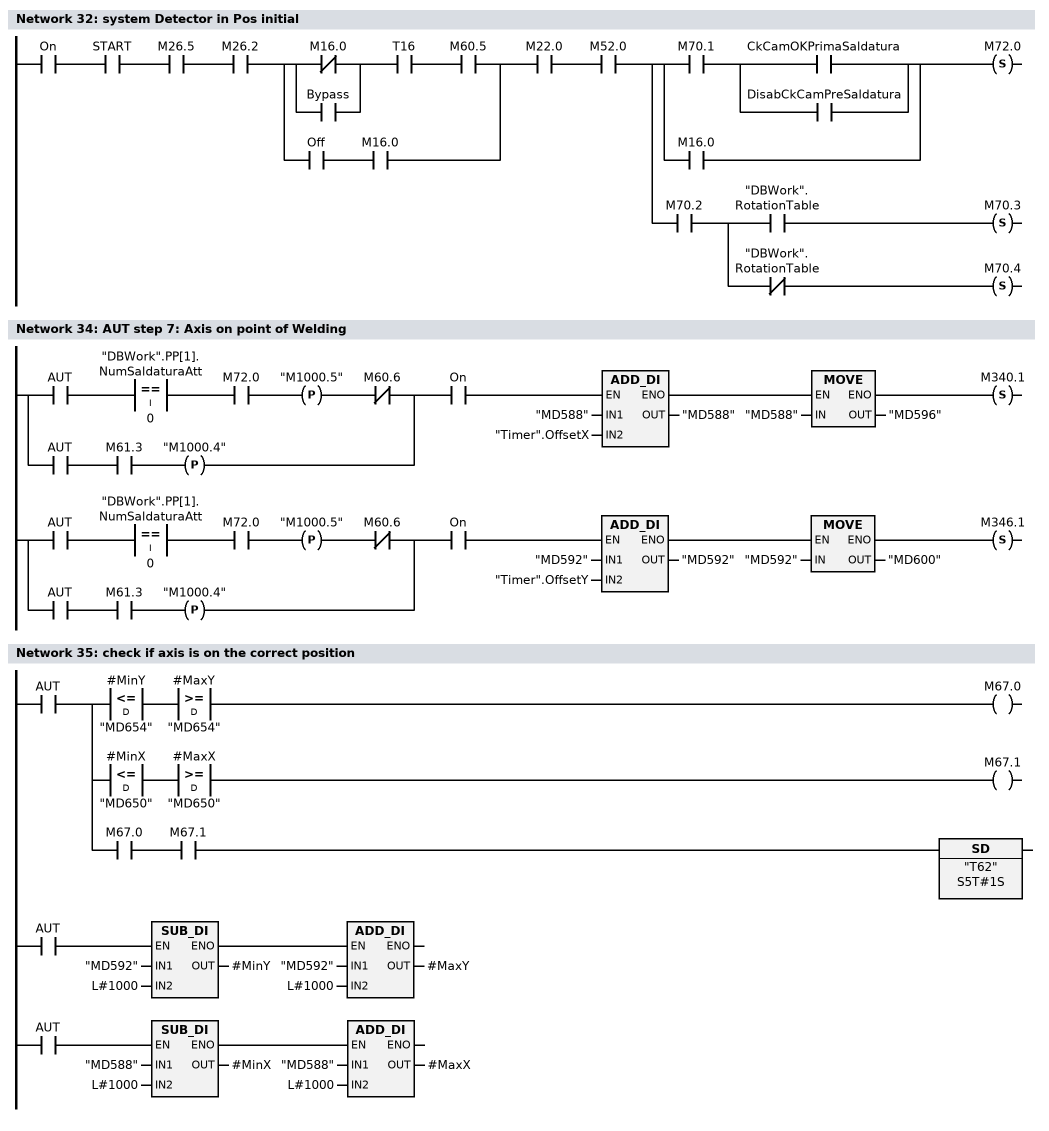
[picture p121: FC14 - AUTOMATIC networks 32-35]
NETWORK
TITLE = system Detector in Pos initial
//System Detector in Pos initial and ready for detect Welding point
      A     "On";
      A     "START";
      A     "M26.5";
      A     "M26.2";
      A(;
      A(;
      ON    "M16.0";
      O     "Bypass";
      );
      A     "T16";
      A     "M60.5";
      O;
      A     "Off";
      A     "M16.0";
      );
      A     "M22.0";
      A     "M52.0";
      =     L 16.0;
      A     L 16.0;
      A(;
      A     "M70.1";
      A(;
      O     "CkCamOKPrimaSaldatura";
      O     "DisabCkCamPreSaldatura";
      );
      O     "M16.0";
      );
      S     "M72.0";
      A     L 16.0;
      A     "M70.2";
      =     L 16.1;
      A     L 16.1;
      A     "DBWork".RotationTable;
      S     "M70.3";
      A     L 16.1;
      AN    "DBWork".RotationTable;
      S     "M70.4";
NETWORK
TITLE = ------------START WITH WELDING
NETWORK
TITLE = AUT step 7: Axis on point of Welding
//AXIS X 
//AXIS Y 
//
//MD588 = SUPPORT FOR POINT X
//MD592 = SUPPORT FOR POINT Y
      A(;
      A     "AUT";
      A(;
      L     "DBWork".PP[1].NumSaldaturaAtt;
      L     0;
      ==I;
      );
      A     "M72.0";
      FP    "M1000.5";
      AN    "M60.6";
      O(;
      A     "AUT";
      A     "M61.3";
      FP    "M1000.4";
      );
      );
      A     "On";
      =     L 16.0;
      A(;
      A     L 16.0;
      JNB   _018;
      L     "MD588";
      L     "Timer".OffsetX;
      +D;
      T     "MD588";
      AN    OV;
      SAVE;
      CLR;
_018: A     BR;
      );
      JNB   _019;
      L     "MD588";
      T     "MD596";
      SET;
      SAVE;
      CLR;
_019: A     BR;
      S     "M340.1";
      A(;
      A     L 16.0;
      JNB   _01a;
      L     "MD592";
      L     "Timer".OffsetY;
      +D;
      T     "MD592";
      AN    OV;
      SAVE;
      CLR;
_01a: A     BR;
      );
      JNB   _01b;
      L     "MD592";
      T     "MD600";
      SET;
      SAVE;
      CLR;
_01b: A     BR;
      S     "M346.1";
NETWORK
TITLE = check if axis is on the correct position
      A     "AUT";
      =     L 16.0;
      A(;
      A     L 16.0;
      JNB   _01c;
      L     "MD592";
      L     L#1000;
      -D;
      T     #MinY;
      AN    OV;
      SAVE;
      CLR;
_01c: A     BR;
      );
      JNB   _01d;
      L     "MD592";
      L     L#1000;
      +D;
      T     #MaxY;
_01d: NOP   0;
      A(;
      A     L 16.0;
      JNB   _01e;
      L     "MD588";
      L     L#1000;
      -D;
      T     #MinX;
      AN    OV;
      SAVE;
      CLR;
_01e: A     BR;
      );
      JNB   _01f;
      L     "MD588";
      L     L#1000;
      +D;
      T     #MaxX;
_01f: NOP   0;
      A     L 16.0;
      A(;
      L     #MinY;
      L     "MD654";
      <=D;
      );
      A(;
      L     #MaxY;
      L     "MD654";
      >=D;
      );
      =     "M67.0";
      A     L 16.0;
      A(;
      L     #MinX;
      L     "MD650";
      <=D;
      );
      A(;
      L     #MaxX;
      L     "MD650";
      >=D;
      );
      =     "M67.1";
      A     L 16.0;
      A     "M67.0";
      A     "M67.1";
      L     S5T#1S;
      SD    "T62";
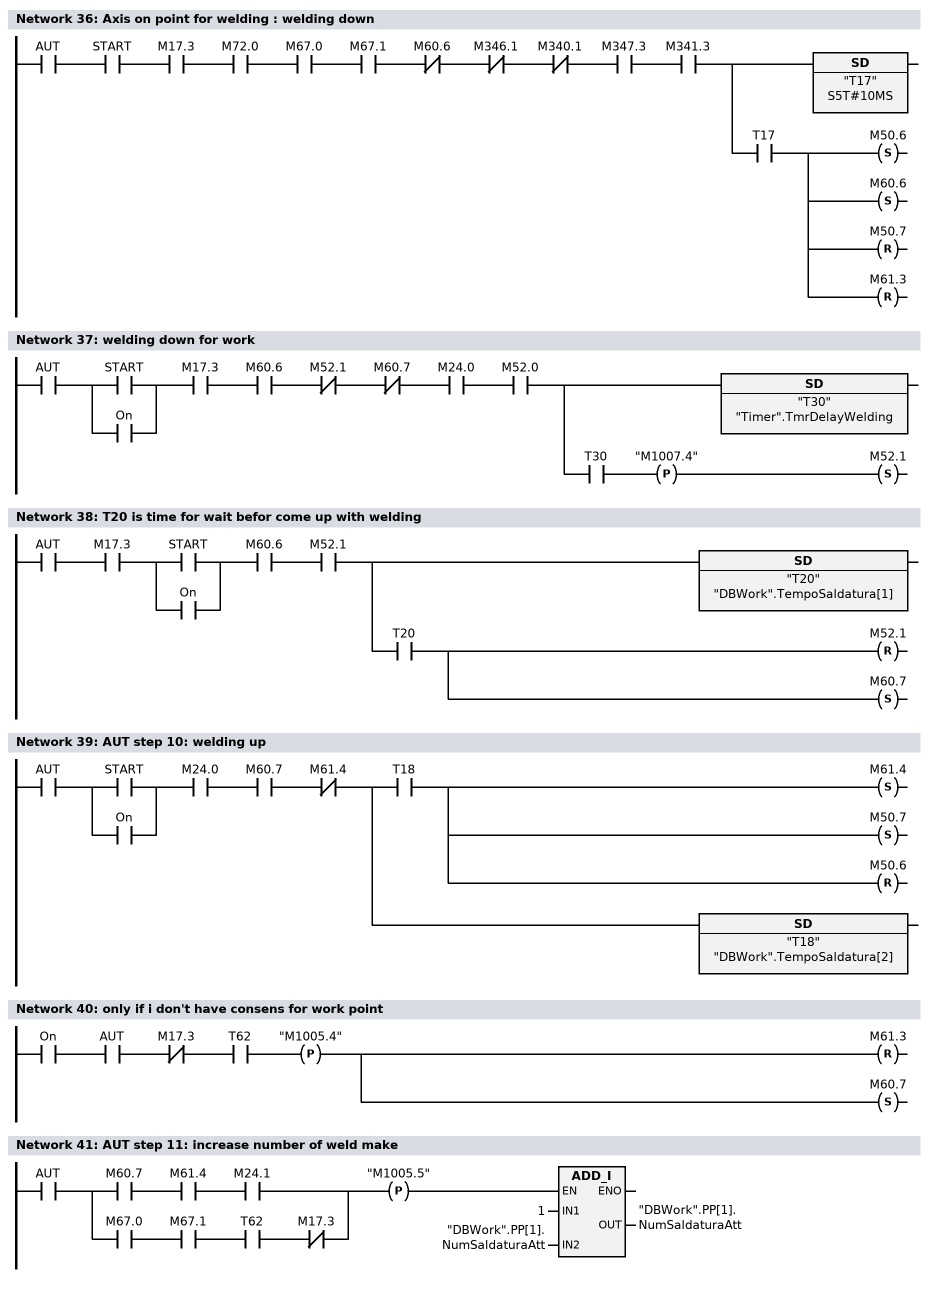
NETWORK
TITLE = Axis on point for welding : welding down
//Saldatore giù
      A     "AUT";
      A     "START";
      A     "M17.3";
      A     "M72.0";
      A     "M67.0";
      A     "M67.1";
      AN    "M60.6";
      AN    "M346.1";
      AN    "M340.1";
      A     "M347.3";
      A     "M341.3";
      =     L 16.0;
      A     L 16.0;
      BLD   102;
      L     S5T#10MS;
      SD    "T17";
      A     L 16.0;
      A     "T17";
      S     "M50.6";
      S     "M60.6";
      R     "M50.7";
      R     "M61.3";
NETWORK
TITLE = welding down for work
//saldatore giu per saldatura
      A     "AUT";
      A(;
      O     "START";
      O     "On";
      );
      A     "M17.3";
      A     "M60.6";
      AN    "M52.1";
      AN    "M60.7";
      A     "M24.0";
      A     "M52.0";
      =     L 16.0;
      A     L 16.0;
      BLD   102;
      L     "Timer".TmrDelayWelding;
      SD    "T30";
      A     L 16.0;
      A     "T30";
      FP    "M1007.4";
      S     "M52.1";
NETWORK
TITLE = T20 is time for wait befor come up with welding
//Resto un tempo T20 sul punto saldato prima di rialzare la torcia
      A     "AUT";
      A     "M17.3";
      A(;
      O     "START";
      O     "On";
      );
      A     "M60.6";
      A     "M52.1";
      =     L 16.0;
      A     L 16.0;
      BLD   102;
      L     "DBWork".TempoSaldatura[1];
      SD    "T20";
      A     L 16.0;
      A     "T20";
      R     "M52.1";
      S     "M60.7";
NETWORK
TITLE = AUT step 10: welding up
      A     "AUT";
      A(;
      O     "START";
      O     "On";
      );
      A     "M24.0";
      A     "M60.7";
      AN    "M61.4";
      =     L 16.0;
      A     L 16.0;
      A     "T18";
      S     "M61.4";
      S     "M50.7";
      R     "M50.6";
      A     L 16.0;
      BLD   102;
      L     "DBWork".TempoSaldatura[2];
      SD    "T18";
NETWORK
TITLE = only if i don't have consens for work point
      A     "On";
      A     "AUT";
      AN    "M17.3";
      A     "T62";
      FP    "M1005.4";
      R     "M61.3";
      S     "M60.7";
NETWORK
TITLE = AUT step 11: increase number of weld make
//incremento il numero di saldature effettuate
      A     "AUT";
      A(;
      A     "M60.7";
      A     "M61.4";
      A     "M24.1";
      O;
      A     "M67.0";
      A     "M67.1";
      A     "T62";
      AN    "M17.3";
      );
      FP    "M1005.5";
      JNB   _020;
      L     1;
      L     "DBWork".PP[1].NumSaldaturaAtt;
      +I;
      T     "DBWork".PP[1].NumSaldaturaAtt;
_020: NOP   0;
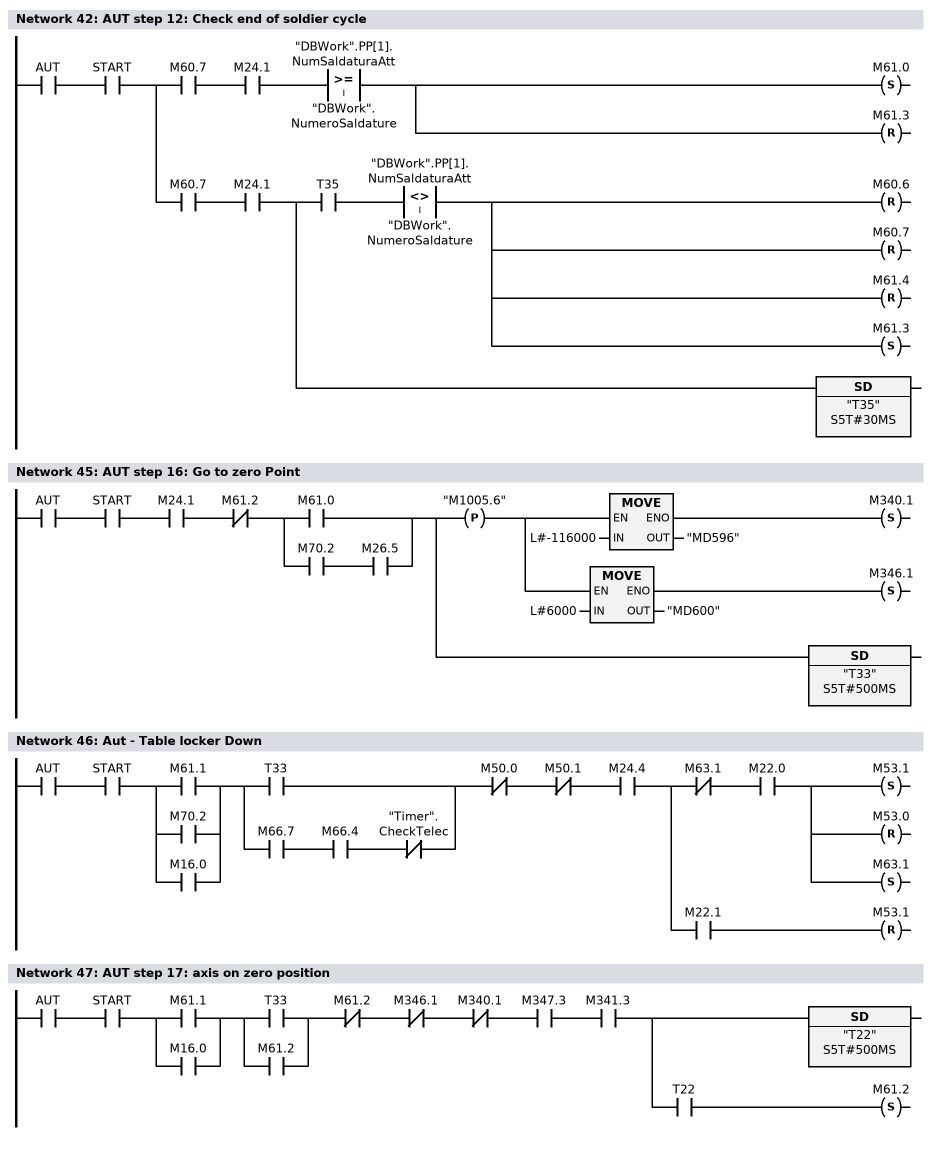
NETWORK
TITLE = AUT step 12: Check end of soldier cycle 
//aspetto per il passaggio delle coorddinate al simodrive
      A     "AUT";
      A     "START";
      =     L 16.0;
      A     L 16.0;
      A     "M60.7";
      A     "M24.1";
      A(;
      L     "DBWork".PP[1].NumSaldaturaAtt;
      L     "DBWork".NumeroSaldature;
      >=I;
      );
      S     "M61.0";
      R     "M61.3";
      A     L 16.0;
      A     "M60.7";
      A     "M24.1";
      =     L 16.1;
      A     L 16.1;
      A     "T35";
      A(;
      L     "DBWork".PP[1].NumSaldaturaAtt;
      L     "DBWork".NumeroSaldature;
      <>I;
      );
      R     "M60.6";
      R     "M60.7";
      R     "M61.4";
      S     "M61.3";
      A     L 16.1;
      BLD   102;
      L     S5T#30MS;
      SD    "T35";
NETWORK
TITLE =
NETWORK
TITLE =
NETWORK
TITLE = AUT step 16: Go to zero Point
      A     "AUT";
      A     "START";
      A     "M24.1";
      AN    "M61.2";
      A(;
      O     "M61.0";
      O;
      A     "M70.2";
      A     "M26.5";
      );
      =     L 16.0;
      A     L 16.0;
      FP    "M1005.6";
      =     L 16.1;
      A     L 16.1;
      JNB   _021;
      L     L#-116000;
      T     "MD596";
      SET;
      SAVE;
      CLR;
_021: A     BR;
      S     "M340.1";
      A     L 16.1;
      JNB   _022;
      L     L#6000;
      T     "MD600";
      SET;
      SAVE;
      CLR;
_022: A     BR;
      S     "M346.1";
      A     L 16.0;
      BLD   102;
      L     S5T#500MS;
      SD    "T33";
NETWORK
TITLE = Aut - Table locker Down
//Table cyclinder Low
      A     "AUT";
      A     "START";
      A(;
      O     "M61.1";
      O     "M70.2";
      O     "M16.0";
      );
      A(;
      O     "T33";
      O;
      A     "M66.7";
      A     "M66.4";
      AN    "Timer".CheckTelec;
      );
      AN    "M50.0";
      AN    "M50.1";
      A     "M24.4";
      =     L 16.0;
      A     L 16.0;
      AN    "M63.1";
      A     "M22.0";
      S     "M53.1";
      R     "M53.0";
      S     "M63.1";
      A     L 16.0;
      A     "M22.1";
      R     "M53.1";
NETWORK
TITLE = AUT step 17: axis on zero position
      A     "AUT";
      A     "START";
      A(;
      O     "M61.1";
      O     "M16.0";
      );
      A(;
      O     "T33";
      O     "M61.2";
      );
      AN    "M61.2";
      AN    "M346.1";
      AN    "M340.1";
      A     "M347.3";
      A     "M341.3";
      =     L 16.0;
      A     L 16.0;
      BLD   102;
      L     S5T#500MS;
      SD    "T22";
      A     L 16.0;
      A     "T22";
      S     "M61.2";
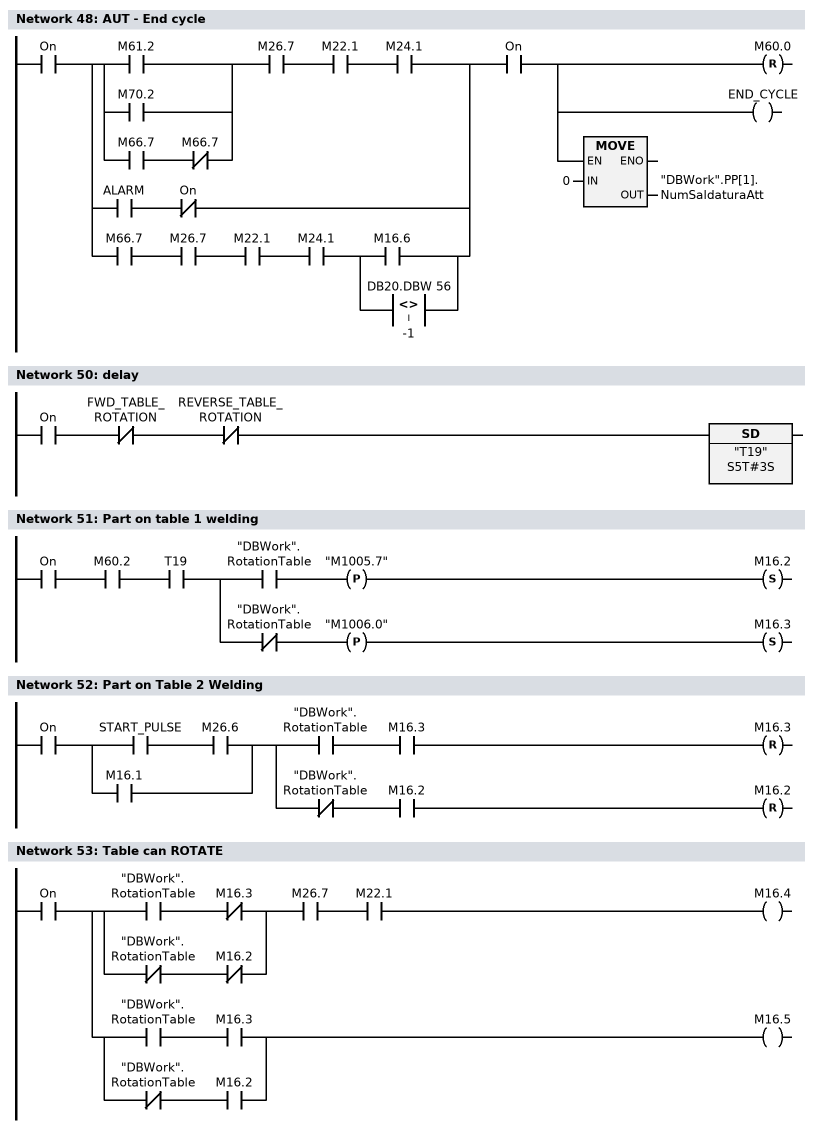
NETWORK
TITLE = AUT - End cycle
      A     "On";
      A(;
      A(;
      O     "M61.2";
      O     "M70.2";
      O;
      A     "M66.7";
      AN    "M66.7";
      );
      A     "M26.7";
      A     "M22.1";
      A     "M24.1";
      O;
      A     "ALARM";
      AN    "On";
      O;
      A     "M66.7";
      A     "M26.7";
      A     "M22.1";
      A     "M24.1";
      A(;
      O     "M16.6";
      O(;
      L     DB20.DBW 56;
      L     -1;
      <>I;
      );
      );
      );
      A     "On";
      =     L 16.0;
      A     L 16.0;
      BLD   102;
      R     "M60.0";
      A     L 16.0;
      BLD   102;
      =     "END_CYCLE";
      A     L 16.0;
      JNB   _023;
      L     0;
      T     "DBWork".PP[1].NumSaldaturaAtt;
_023: NOP   0;
NETWORK
TITLE =
NETWORK
TITLE = delay
      A     "On";
      AN    "FWD_TABLE_ROTATION";
      AN    "REVERSE_TABLE_ROTATION";
      L     S5T#3S;
      SD    "T19";
NETWORK
TITLE = Part on table 1 welding
      A     "On";
      A     "M60.2";
      A     "T19";
      =     L 16.0;
      A     L 16.0;
      A     "DBWork".RotationTable;
      FP    "M1005.7";
      S     "M16.2";
      A     L 16.0;
      AN    "DBWork".RotationTable;
      FP    "M1006.0";
      S     "M16.3";
NETWORK
TITLE = Part on Table 2 Welding
      A     "On";
      A(;
      A     "START_PULSE";
      A     "M26.6";
      O     "M16.1";
      );
      =     L 16.0;
      A     L 16.0;
      A     "DBWork".RotationTable;
      A     "M16.3";
      R     "M16.3";
      A     L 16.0;
      AN    "DBWork".RotationTable;
      A     "M16.2";
      R     "M16.2";
NETWORK
TITLE = Table can ROTATE
      A     "On";
      =     L 16.0;
      A     L 16.0;
      A(;
      A     "DBWork".RotationTable;
      AN    "M16.3";
      O;
      AN    "DBWork".RotationTable;
      AN    "M16.2";
      );
      A     "M26.7";
      A     "M22.1";
      =     "M16.4";
      A     L 16.0;
      A(;
      A     "DBWork".RotationTable;
      A     "M16.3";
      O;
      AN    "DBWork".RotationTable;
      A     "M16.2";
      );
      =     "M16.5";
END_FUNCTION

FUNCTION "FC16 - ALARMS" : VOID	// FC 16
TITLE = Alarms management
VERSION : 0.1
VAR_TEMP
  tempBOOL : BOOL ;
END_VAR
BEGIN
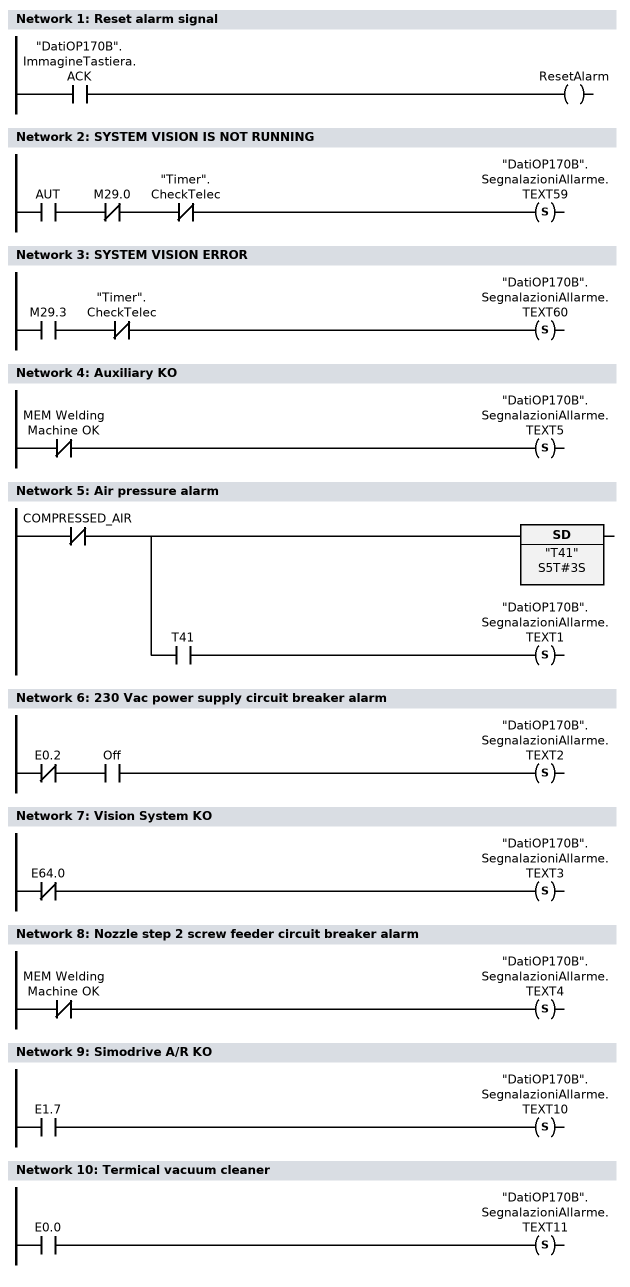
NETWORK
TITLE = Reset alarm signal
      A     "DatiOP170B".ImmagineTastiera.ACK;
      =     "ResetAlarm";
NETWORK
TITLE = SYSTEM VISION IS NOT RUNNING
      A     "AUT";
      AN    "M29.0";
      AN    "Timer".CheckTelec;
      S     "DatiOP170B".SegnalazioniAllarme.TEXT59;
NETWORK
TITLE = SYSTEM VISION ERROR
      A     "M29.3";
      AN    "Timer".CheckTelec;
      S     "DatiOP170B".SegnalazioniAllarme.TEXT60;
NETWORK
TITLE = Auxiliary KO
      AN    "MEM Welding Machine OK";
      S     "DatiOP170B".SegnalazioniAllarme.TEXT5;
NETWORK
TITLE = Air pressure alarm
      AN    "COMPRESSED_AIR";
      =     L 1.0;
      A     L 1.0;
      BLD   102;
      L     S5T#3S;
      SD    "T41";
      A     L 1.0;
      A     "T41";
      S     "DatiOP170B".SegnalazioniAllarme.TEXT1;
NETWORK
TITLE = 230 Vac power supply circuit breaker alarm
      AN    "E0.2";
      A     "Off";
      S     "DatiOP170B".SegnalazioniAllarme.TEXT2;
NETWORK
TITLE = Vision System KO
      AN    "E64.0";
      S     "DatiOP170B".SegnalazioniAllarme.TEXT3;
NETWORK
TITLE = Nozzle step 2 screw feeder circuit breaker alarm
      AN    "MEM Welding Machine OK";
      S     "DatiOP170B".SegnalazioniAllarme.TEXT4;
NETWORK
TITLE = Simodrive A/R KO
      A     "E1.7";
      S     "DatiOP170B".SegnalazioniAllarme.TEXT10;
NETWORK
TITLE = Termical vacuum cleaner
      A     "E0.0";
      S     "DatiOP170B".SegnalazioniAllarme.TEXT11;
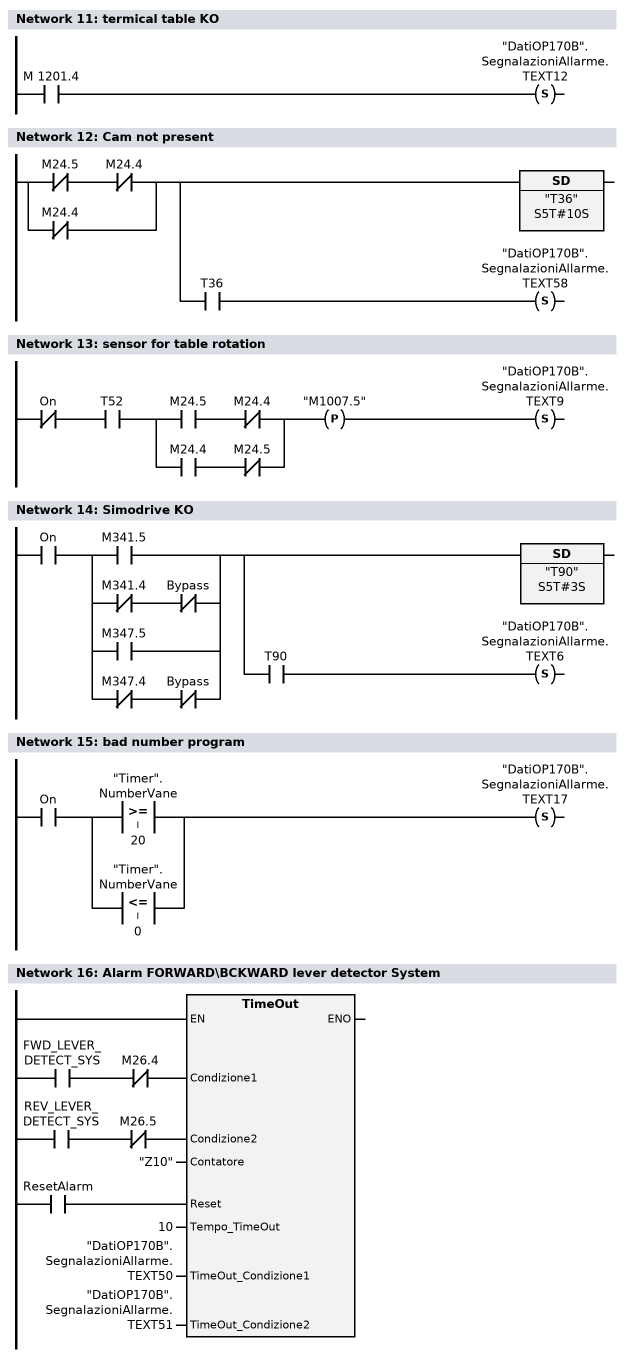
NETWORK
TITLE = termical table KO
      A     M 1201.4;
      S     "DatiOP170B".SegnalazioniAllarme.TEXT12;
NETWORK
TITLE = Cam not present
      AN    "M24.5";
      AN    "M24.4";
      ON    "M24.4";
      =     L 1.0;
      A     L 1.0;
      BLD   102;
      L     S5T#10S;
      SD    "T36";
      A     L 1.0;
      A     "T36";
      S     "DatiOP170B".SegnalazioniAllarme.TEXT58;
NETWORK
TITLE = sensor for table rotation
      AN    "On";
      A     "T52";
      A(;
      A     "M24.5";
      AN    "M24.4";
      O;
      A     "M24.4";
      AN    "M24.5";
      );
      FP    "M1007.5";
      S     "DatiOP170B".SegnalazioniAllarme.TEXT9;
NETWORK
TITLE = Simodrive KO
//press ack button
      A     "On";
      A(;
      O     "M341.5";
      O;
      AN    "M341.4";
      AN    "Bypass";
      O     "M347.5";
      O;
      AN    "M347.4";
      AN    "Bypass";
      );
      =     L 1.0;
      A     L 1.0;
      BLD   102;
      L     S5T#3S;
      SD    "T90";
      A     L 1.0;
      A     "T90";
      S     "DatiOP170B".SegnalazioniAllarme.TEXT6;
NETWORK
TITLE = bad number program
      A     "On";
      A(;
      O(;
      L     "Timer".NumberVane;
      L     20;
      >=I;
      );
      O(;
      L     "Timer".NumberVane;
      L     0;
      <=I;
      );
      );
      S     "DatiOP170B".SegnalazioniAllarme.TEXT17;
NETWORK
TITLE = Alarm FORWARD\BCKWARD lever detector System
      A     "FWD_LEVER_DETECT_SYS";
      AN    "M26.4";
      =     L 1.0;
      BLD   103;
      A     "REV_LEVER_DETECT_SYS";
      AN    "M26.5";
      =     L 1.1;
      BLD   103;
      A     "ResetAlarm";
      =     L 1.2;
      BLD   103;
      CALL  "TimeOut" (
           Condizione1              := L 1.0,
           Condizione2              := L 1.1,
           Contatore                := "Z10",
           Reset                    := L 1.2,
           Tempo_TimeOut            := 10,
           TimeOut_Condizione1      := "DatiOP170B".SegnalazioniAllarme.TEXT50,
           TimeOut_Condizione2      := "DatiOP170B".SegnalazioniAllarme.TEXT51);
      NOP   0;
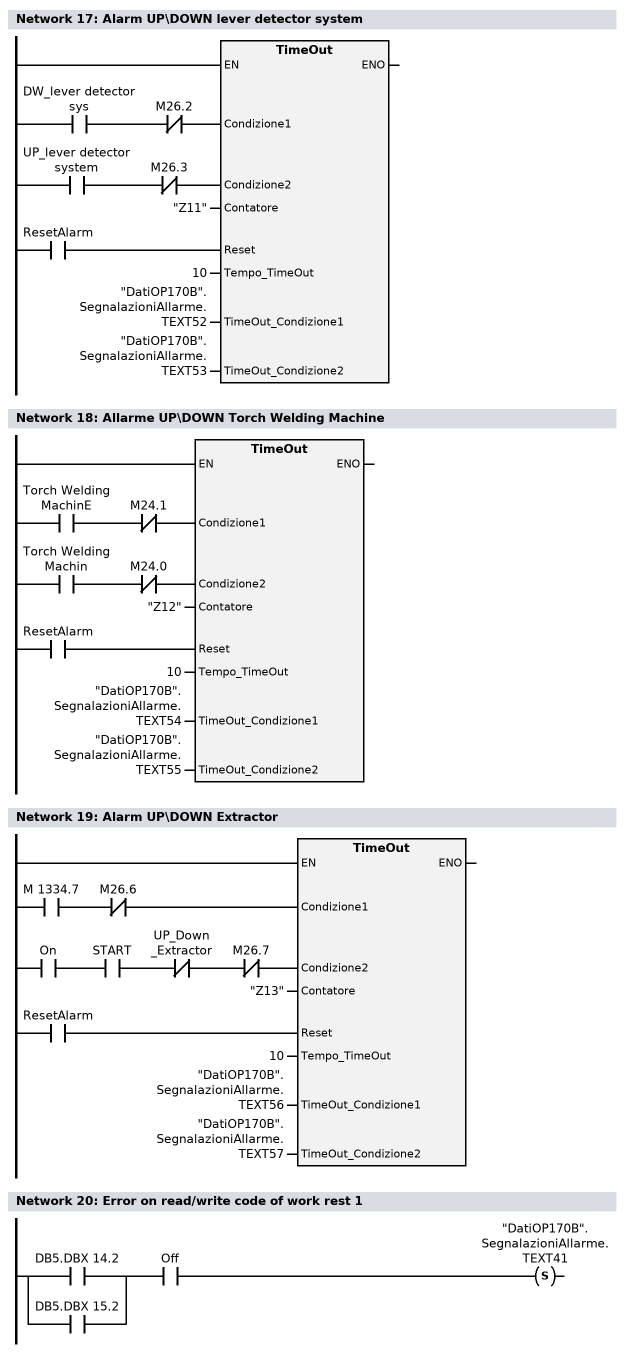
NETWORK
TITLE = Alarm UP\DOWN lever detector system
      A     "DW_lever detector sys";
      AN    "M26.2";
      =     L 1.0;
      BLD   103;
      A     "UP_lever detector system";
      AN    "M26.3";
      =     L 1.1;
      BLD   103;
      A     "ResetAlarm";
      =     L 1.2;
      BLD   103;
      CALL  "TimeOut" (
           Condizione1              := L 1.0,
           Condizione2              := L 1.1,
           Contatore                := "Z11",
           Reset                    := L 1.2,
           Tempo_TimeOut            := 10,
           TimeOut_Condizione1      := "DatiOP170B".SegnalazioniAllarme.TEXT52,
           TimeOut_Condizione2      := "DatiOP170B".SegnalazioniAllarme.TEXT53);
      NOP   0;
NETWORK
TITLE = Allarme UP\DOWN Torch Welding Machine
      A     "Torch Welding MachinE";
      AN    "M24.1";
      =     L 1.0;
      BLD   103;
      A     "Torch Welding Machin";
      AN    "M24.0";
      =     L 1.1;
      BLD   103;
      A     "ResetAlarm";
      =     L 1.2;
      BLD   103;
      CALL  "TimeOut" (
           Condizione1              := L 1.0,
           Condizione2              := L 1.1,
           Contatore                := "Z12",
           Reset                    := L 1.2,
           Tempo_TimeOut            := 10,
           TimeOut_Condizione1      := "DatiOP170B".SegnalazioniAllarme.TEXT54,
           TimeOut_Condizione2      := "DatiOP170B".SegnalazioniAllarme.TEXT55);
      NOP   0;
NETWORK
TITLE = Alarm UP\DOWN Extractor
      A     M 1334.7;
      AN    "M26.6";
      =     L 1.0;
      BLD   103;
      A     "On";
      A     "START";
      AN    "UP_Down _Extractor";
      AN    "M26.7";
      =     L 1.1;
      BLD   103;
      A     "ResetAlarm";
      =     L 1.2;
      BLD   103;
      CALL  "TimeOut" (
           Condizione1              := L 1.0,
           Condizione2              := L 1.1,
           Contatore                := "Z13",
           Reset                    := L 1.2,
           Tempo_TimeOut            := 10,
           TimeOut_Condizione1      := "DatiOP170B".SegnalazioniAllarme.TEXT56,
           TimeOut_Condizione2      := "DatiOP170B".SegnalazioniAllarme.TEXT57);
      NOP   0;
NETWORK
TITLE = Error on read/write code of work rest 1
      A(;
      O     DB5.DBX 14.2;
      O     DB5.DBX 15.2;
      );
      A     "Off";
      S     "DatiOP170B".SegnalazioniAllarme.TEXT41;
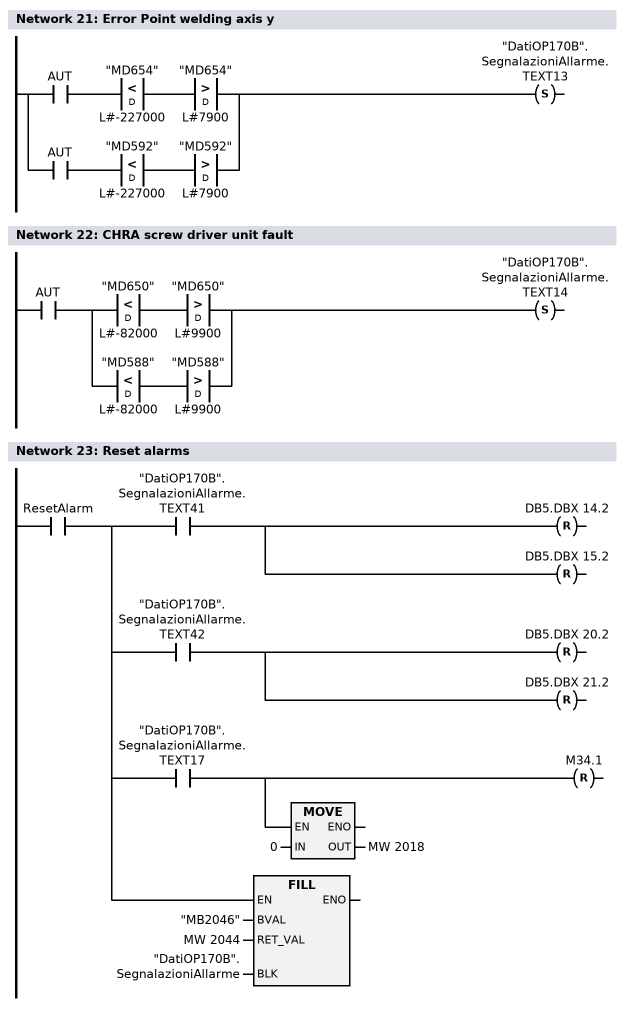
NETWORK
TITLE = Error Point welding axis y
      A     "AUT";
      A(;
      L     "MD654";
      L     L#-227000;
      <D;
      );
      A(;
      L     "MD654";
      L     L#7900;
      >D;
      );
      O;
      A     "AUT";
      A(;
      L     "MD592";
      L     L#-227000;
      <D;
      );
      A(;
      L     "MD592";
      L     L#7900;
      >D;
      );
      S     "DatiOP170B".SegnalazioniAllarme.TEXT13;
NETWORK
TITLE = CHRA screw driver unit fault
      A     "AUT";
      A(;
      A(;
      L     "MD650";
      L     L#-82000;
      <D;
      );
      A(;
      L     "MD650";
      L     L#9900;
      >D;
      );
      O;
      A(;
      L     "MD588";
      L     L#-82000;
      <D;
      );
      A(;
      L     "MD588";
      L     L#9900;
      >D;
      );
      );
      S     "DatiOP170B".SegnalazioniAllarme.TEXT14;
NETWORK
TITLE = Reset alarms
      A     "ResetAlarm";
      =     L 1.0;
      A     L 1.0;
      A     "DatiOP170B".SegnalazioniAllarme.TEXT41;
      R     DB5.DBX 14.2;
      R     DB5.DBX 15.2;
      A     L 1.0;
      A     "DatiOP170B".SegnalazioniAllarme.TEXT42;
      R     DB5.DBX 20.2;
      R     DB5.DBX 21.2;
      A     L 1.0;
      A     "DatiOP170B".SegnalazioniAllarme.TEXT17;
      =     L 1.1;
      A     L 1.1;
      BLD   102;
      R     "M34.1";
      A     L 1.1;
      JNB   _001;
      L     0;
      T     MW 2018;
_001: NOP   0;
      A     L 1.0;
      JNB   _002;
      CALL  "FILL" (
           BVAL                     := "MB2046",
           RET_VAL                  := MW 2044,
           BLK                      := "DatiOP170B".SegnalazioniAllarme);
_002: NOP   0;
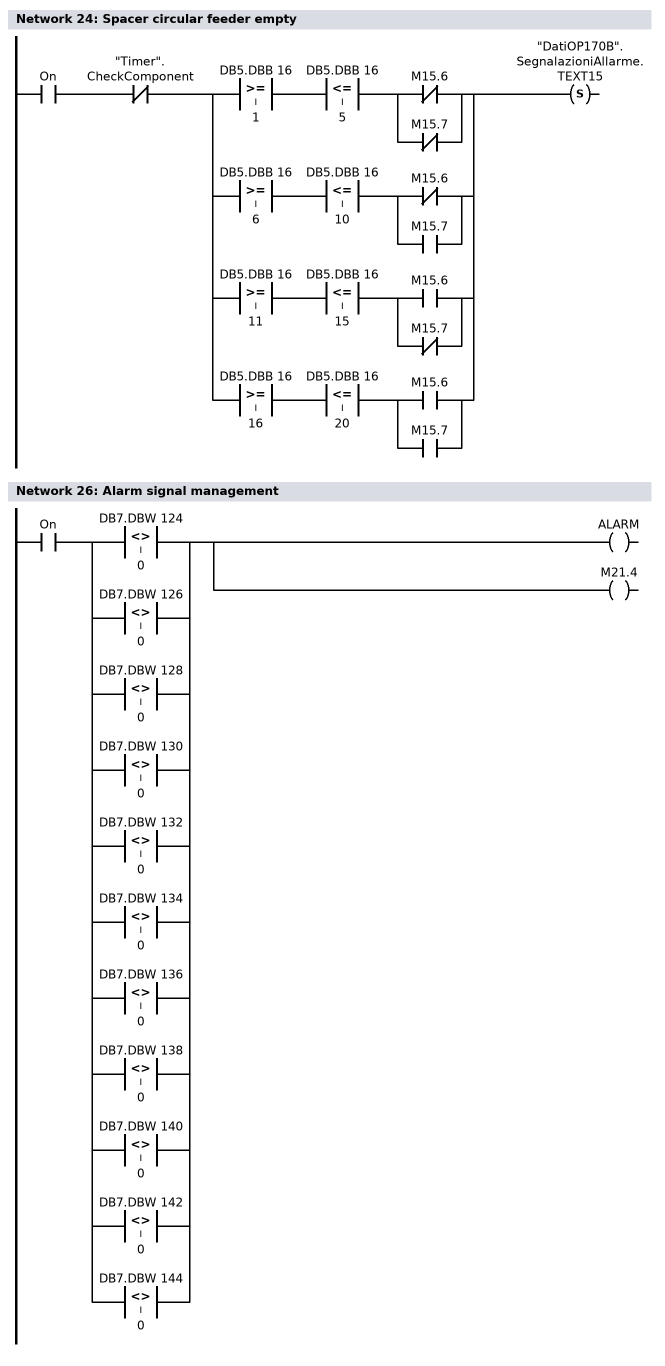
NETWORK
TITLE = Spacer circular feeder empty
      A     "On";
      AN    "Timer".CheckComponent;
      A(;
      A(;
      L     DB5.DBB 16;
      L     1;
      >=I;
      );
      A(;
      L     DB5.DBB 16;
      L     5;
      <=I;
      );
      A(;
      ON    "M15.6";
      ON    "M15.7";
      );
      O;
      A(;
      L     DB5.DBB 16;
      L     6;
      >=I;
      );
      A(;
      L     DB5.DBB 16;
      L     10;
      <=I;
      );
      A(;
      ON    "M15.6";
      O     "M15.7";
      );
      O;
      A(;
      L     DB5.DBB 16;
      L     11;
      >=I;
      );
      A(;
      L     DB5.DBB 16;
      L     15;
      <=I;
      );
      A(;
      O     "M15.6";
      ON    "M15.7";
      );
      O;
      A(;
      L     DB5.DBB 16;
      L     16;
      >=I;
      );
      A(;
      L     DB5.DBB 16;
      L     20;
      <=I;
      );
      A(;
      O     "M15.6";
      O     "M15.7";
      );
      );
      S     "DatiOP170B".SegnalazioniAllarme.TEXT15;
NETWORK
TITLE =
      A     "On";
      A(;
      A(;
      L     "Timer".NumberVane;
      L     1;
      >=I;
      );
      A(;
      L     "Timer".NumberVane;
      L     5;
      <=I;
      );
      A(;
      O(;
      L     DB5.DBB 16;
      L     1;
      <I;
      );
      O(;
      L     DB5.DBB 16;
      L     5;
      >I;
      );
      );
      O;
      A(;
      L     "Timer".NumberVane;
      L     6;
      >=I;
      );
      A(;
      L     "Timer".NumberVane;
      L     10;
      <=I;
      );
      A(;
      O(;
      L     DB5.DBB 16;
      L     6;
      <I;
      );
      O(;
      L     DB5.DBB 16;
      L     10;
      >I;
      );
      );
      O;
      A(;
      L     "Timer".NumberVane;
      L     11;
      >=I;
      );
      A(;
      L     "Timer".NumberVane;
      L     15;
      <=I;
      );
      A(;
      O(;
      L     DB5.DBB 16;
      L     11;
      <I;
      );
      O(;
      L     DB5.DBB 16;
      L     15;
      >I;
      );
      );
      O;
      A(;
      L     "Timer".NumberVane;
      L     16;
      >=I;
      );
      A(;
      L     "Timer".NumberVane;
      L     20;
      <=I;
      );
      A(;
      O(;
      L     DB5.DBB 16;
      L     16;
      <I;
      );
      O(;
      L     DB5.DBB 16;
      L     20;
      >I;
      );
      );
      );
//   S     "DatiOP170B".SegnalazioniAllarme.TEXT16
NETWORK
TITLE = Alarm signal management
      A     "On";
      A(;
      O(;
      L     DB7.DBW 124;
      L     0;
      <>I;
      );
      O(;
      L     DB7.DBW 126;
      L     0;
      <>I;
      );
      O(;
      L     DB7.DBW 128;
      L     0;
      <>I;
      );
      O(;
      L     DB7.DBW 130;
      L     0;
      <>I;
      );
      O(;
      L     DB7.DBW 132;
      L     0;
      <>I;
      );
      O(;
      L     DB7.DBW 134;
      L     0;
      <>I;
      );
      O(;
      L     DB7.DBW 136;
      L     0;
      <>I;
      );
      O(;
      L     DB7.DBW 138;
      L     0;
      <>I;
      );
      O(;
      L     DB7.DBW 140;
      L     0;
      <>I;
      );
      O(;
      L     DB7.DBW 142;
      L     0;
      <>I;
      );
      O(;
      L     DB7.DBW 144;
      L     0;
      <>I;
      );
      );
      =     "ALARM";
      =     "M21.4";
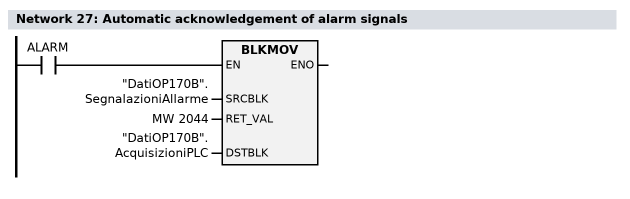
NETWORK
TITLE = Automatic acknowledgement of alarm signals
      A     "ALARM";
      JNB   _003;
      CALL  "BLKMOV" (
           SRCBLK                   := "DatiOP170B".SegnalazioniAllarme,
           RET_VAL                  := MW 2044,
           DSTBLK                   := "DatiOP170B".AcquisizioniPLC);
_003: NOP   0;
END_FUNCTION

FUNCTION "FC17 - OPERATOR PANNEL" : VOID	// FC 17
TITLE = OP170B Operator Pannel Interface
VERSION : 0.1
BEGIN
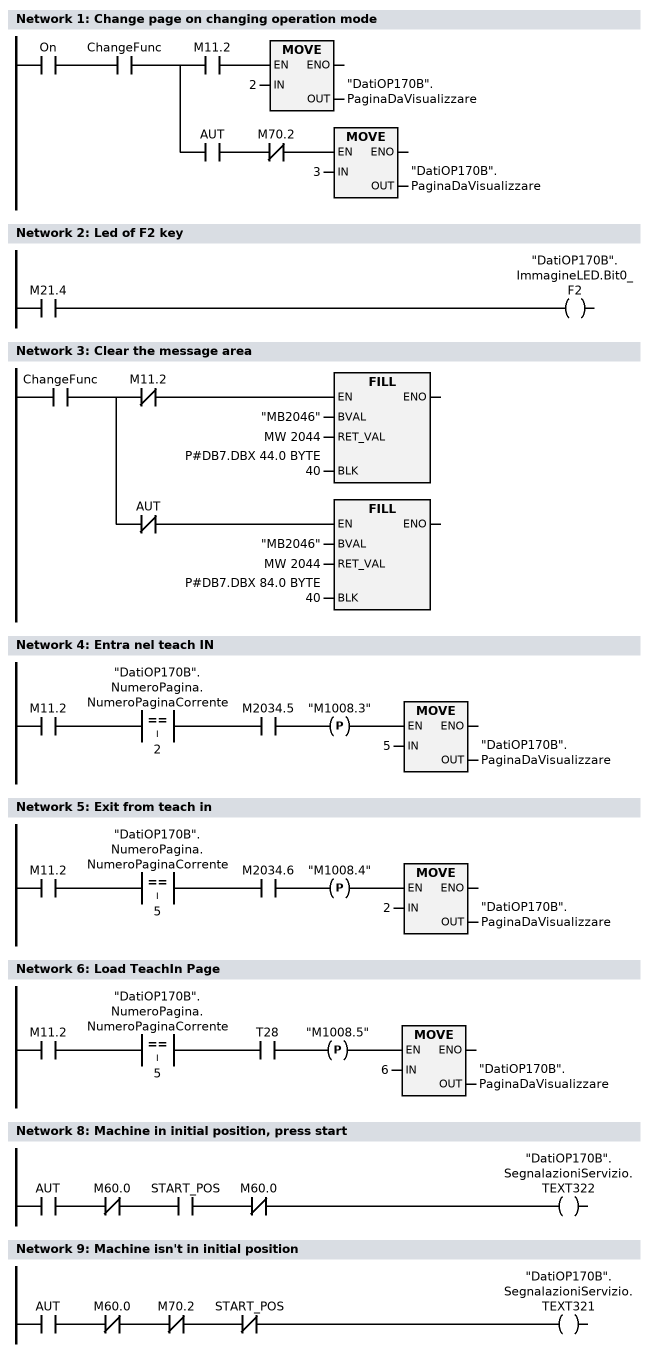
NETWORK
TITLE = Change page on changing operation mode
      A     "On";
      A     "ChangeFunc";
      =     L 0.0;
      A     L 0.0;
      A     "M11.2";
      JNB   _001;
      L     2;
      T     "DatiOP170B".PaginaDaVisualizzare;
_001: NOP   0;
      A     L 0.0;
      A     "AUT";
      AN    "M70.2";
      JNB   _002;
      L     3;
      T     "DatiOP170B".PaginaDaVisualizzare;
_002: NOP   0;
NETWORK
TITLE = Led of F2 key
      A     "M21.4";
      =     "DatiOP170B".ImmagineLED.Bit0_F2;
NETWORK
TITLE = Clear the message area
      A     "ChangeFunc";
      =     L 0.0;
      A     L 0.0;
      AN    "M11.2";
      JNB   _003;
      CALL  "FILL" (
           BVAL                     := "MB2046",
           RET_VAL                  := MW 2044,
           BLK                      := P#DB7.DBX 44.0 BYTE 40);
_003: NOP   0;
      A     L 0.0;
      AN    "AUT";
      JNB   _004;
      CALL  "FILL" (
           BVAL                     := "MB2046",
           RET_VAL                  := MW 2044,
           BLK                      := P#DB7.DBX 84.0 BYTE 40);
_004: NOP   0;
NETWORK
TITLE = Entra nel teach IN
      A     "M11.2";
      A(;
      L     "DatiOP170B".NumeroPagina.NumeroPaginaCorrente;
      L     2;
      ==I;
      );
      A     "M2034.5";
      FP    "M1008.3";
      JNB   _005;
      L     5;
      T     "DatiOP170B".PaginaDaVisualizzare;
_005: NOP   0;
NETWORK
TITLE = Exit from teach in
      A     "M11.2";
      A(;
      L     "DatiOP170B".NumeroPagina.NumeroPaginaCorrente;
      L     5;
      ==I;
      );
      A     "M2034.6";
      FP    "M1008.4";
      JNB   _006;
      L     2;
      T     "DatiOP170B".PaginaDaVisualizzare;
_006: NOP   0;
NETWORK
TITLE = Load TeachIn Page
//Aspetto il T28 in modo tale da lanciare il comando agli assi
      A     "M11.2";
      A(;
      L     "DatiOP170B".NumeroPagina.NumeroPaginaCorrente;
      L     5;
      ==I;
      );
      A     "T28";
      FP    "M1008.5";
      JNB   _007;
      L     6;
      T     "DatiOP170B".PaginaDaVisualizzare;
_007: NOP   0;
NETWORK
TITLE =
NETWORK
TITLE = Machine in initial position, press start
      A     "AUT";
      AN    "M60.0";
      A     "START_POS";
      AN    "M60.0";
      =     "DatiOP170B".SegnalazioniServizio.TEXT322;
NETWORK
TITLE = Machine isn't in initial position
      A     "AUT";
      AN    "M60.0";
      AN    "M70.2";
      AN    "START_POS";
      =     "DatiOP170B".SegnalazioniServizio.TEXT321;
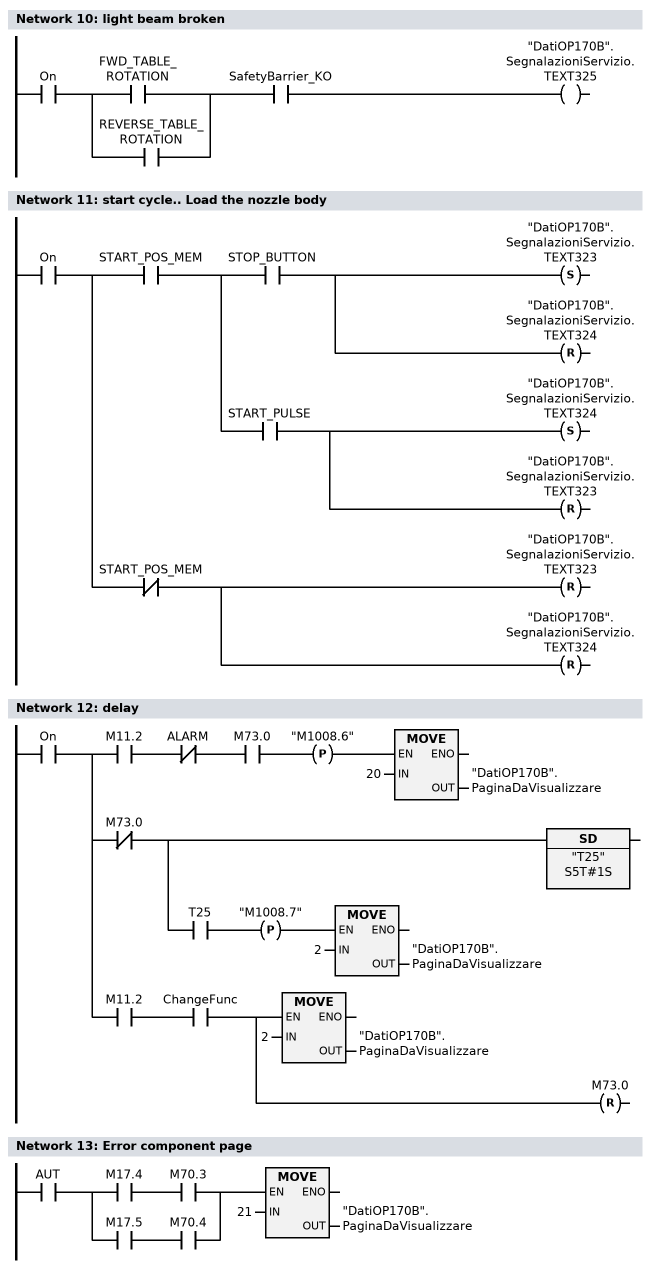
NETWORK
TITLE = light beam broken
      A     "On";
      A(;
      O     "FWD_TABLE_ROTATION";
      O     "REVERSE_TABLE_ROTATION";
      );
      A     "SafetyBarrier_KO";
      =     "DatiOP170B".SegnalazioniServizio.TEXT325;
NETWORK
TITLE = start cycle.. Load the nozzle body
      A     "On";
      =     L 0.0;
      A     L 0.0;
      A     "START_POS_MEM";
      =     L 0.1;
      A     L 0.1;
      A     "STOP_BUTTON";
      S     "DatiOP170B".SegnalazioniServizio.TEXT323;
      R     "DatiOP170B".SegnalazioniServizio.TEXT324;
      A     L 0.1;
      A     "START_PULSE";
      S     "DatiOP170B".SegnalazioniServizio.TEXT324;
      R     "DatiOP170B".SegnalazioniServizio.TEXT323;
      A     L 0.0;
      AN    "START_POS_MEM";
      R     "DatiOP170B".SegnalazioniServizio.TEXT323;
      R     "DatiOP170B".SegnalazioniServizio.TEXT324;
NETWORK
TITLE = delay
//Page of repositioning
      A     "On";
      =     L 0.0;
      A     L 0.0;
      A     "M11.2";
      AN    "ALARM";
      A     "M73.0";
      FP    "M1008.6";
      JNB   _008;
      L     20;
      T     "DatiOP170B".PaginaDaVisualizzare;
_008: NOP   0;
      A     L 0.0;
      AN    "M73.0";
      =     L 0.1;
      A     L 0.1;
      BLD   102;
      L     S5T#1S;
      SD    "T25";
      A     L 0.1;
      A     "T25";
      FP    "M1008.7";
      JNB   _009;
      L     2;
      T     "DatiOP170B".PaginaDaVisualizzare;
_009: NOP   0;
      A     L 0.0;
      A     "M11.2";
      A     "ChangeFunc";
      =     L 0.1;
      A     L 0.1;
      JNB   _00a;
      L     2;
      T     "DatiOP170B".PaginaDaVisualizzare;
_00a: NOP   0;
      A     L 0.1;
      BLD   102;
      R     "M73.0";
NETWORK
TITLE = Error component page
      A     "AUT";
      A(;
      A     "M17.4";
      A     "M70.3";
      O;
      A     "M17.5";
      A     "M70.4";
      );
      JNB   _00b;
      L     21;
      T     "DatiOP170B".PaginaDaVisualizzare;
_00b: NOP   0;
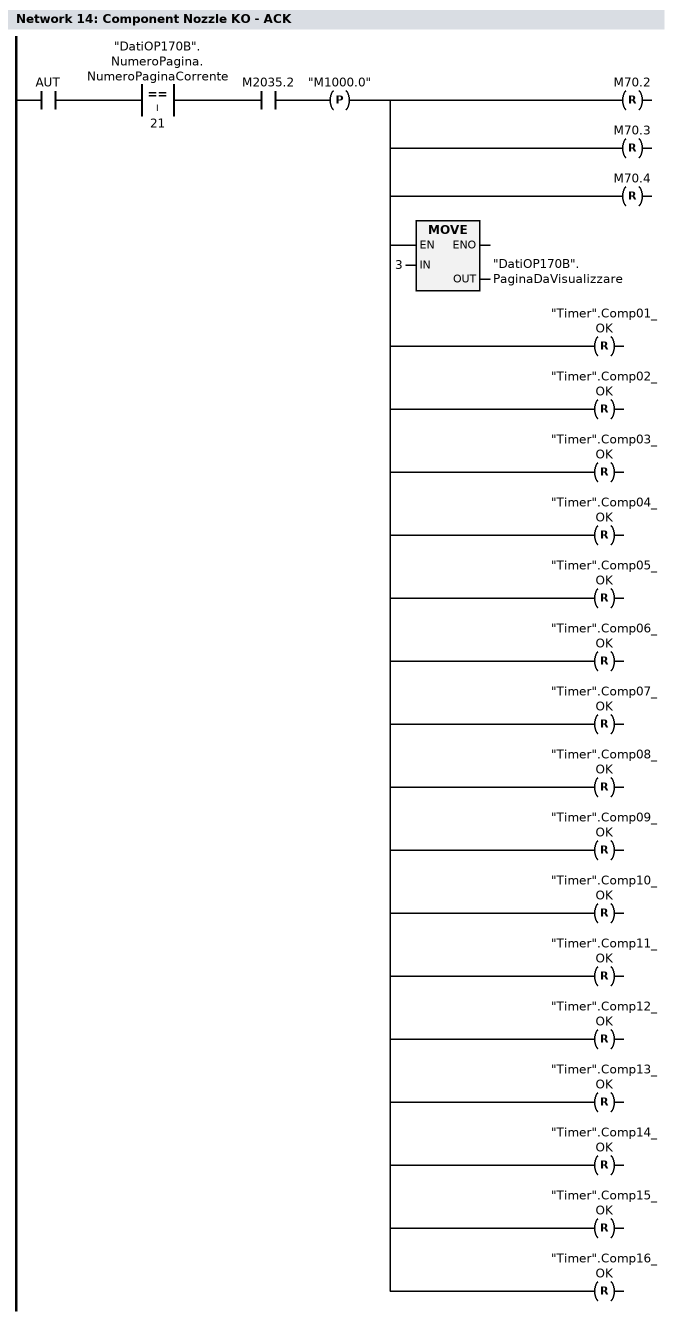
NETWORK
TITLE = Component Nozzle KO - ACK
      A     "AUT";
      A(;
      L     "DatiOP170B".NumeroPagina.NumeroPaginaCorrente;
      L     21;
      ==I;
      );
      A     "M2035.2";
      FP    "M1000.0";
      =     L 0.0;
      A     L 0.0;
      BLD   102;
      R     "M70.2";
      A     L 0.0;
      BLD   102;
      R     "M70.3";
      A     L 0.0;
      BLD   102;
      R     "M70.4";
      A     L 0.0;
      JNB   _00c;
      L     3;
      T     "DatiOP170B".PaginaDaVisualizzare;
_00c: NOP   0;
      A     L 0.0;
      BLD   102;
      R     "Timer".Comp01_OK;
      A     L 0.0;
      BLD   102;
      R     "Timer".Comp02_OK;
      A     L 0.0;
      BLD   102;
      R     "Timer".Comp03_OK;
      A     L 0.0;
      BLD   102;
      R     "Timer".Comp04_OK;
      A     L 0.0;
      BLD   102;
      R     "Timer".Comp05_OK;
      A     L 0.0;
      BLD   102;
      R     "Timer".Comp06_OK;
      A     L 0.0;
      BLD   102;
      R     "Timer".Comp07_OK;
      A     L 0.0;
      BLD   102;
      R     "Timer".Comp08_OK;
      A     L 0.0;
      BLD   102;
      R     "Timer".Comp09_OK;
      A     L 0.0;
      BLD   102;
      R     "Timer".Comp10_OK;
      A     L 0.0;
      BLD   102;
      R     "Timer".Comp11_OK;
      A     L 0.0;
      BLD   102;
      R     "Timer".Comp12_OK;
      A     L 0.0;
      BLD   102;
      R     "Timer".Comp13_OK;
      A     L 0.0;
      BLD   102;
      R     "Timer".Comp14_OK;
      A     L 0.0;
      BLD   102;
      R     "Timer".Comp15_OK;
      A     L 0.0;
      BLD   102;
      R     "Timer".Comp16_OK;
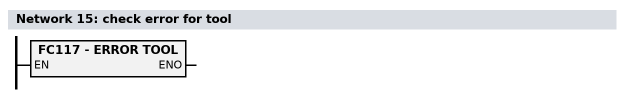
NETWORK
TITLE = check error for tool
      CALL  "FC117 - ERROR TOOL";
      NOP   0;
END_FUNCTION

FUNCTION "FC18 - OUTPUTS" : VOID	// FC 18
TITLE = Outputs management
VERSION : 0.1
BEGIN
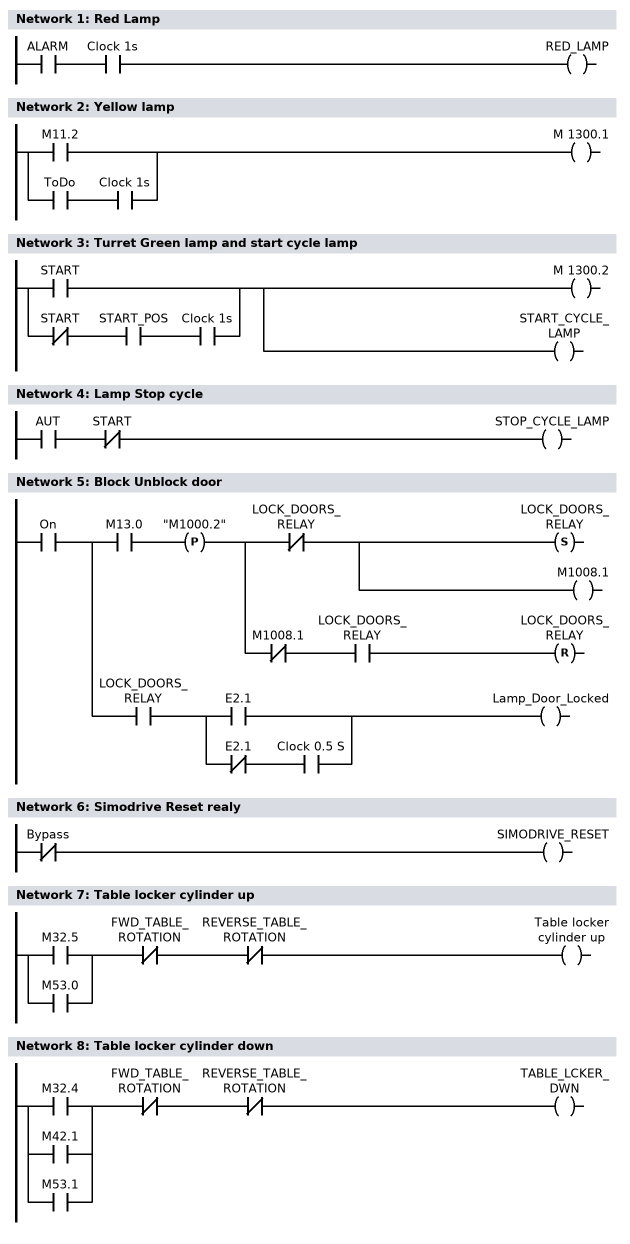
NETWORK
TITLE = Red Lamp
      A     "ALARM";
      A     "Clock 1s";
      =     "RED_LAMP";
NETWORK
TITLE = Yellow lamp
      O     "M11.2";
      O;
      A     "ToDo";
      A     "Clock 1s";
      =     M 1300.1;
NETWORK
TITLE = Turret Green lamp and start cycle lamp
      O     "START";
      O;
      AN    "START";
      A     "START_POS";
      A     "Clock 1s";
      =     M 1300.2;
      =     "START_CYCLE_LAMP";
NETWORK
TITLE = Lamp Stop cycle
      A     "AUT";
      AN    "START";
      =     "STOP_CYCLE_LAMP";
NETWORK
TITLE = Block Unblock door
//light ON = door lock
      A     "On";
      =     L 0.0;
      A     L 0.0;
      A     "M13.0";
      FP    "M1000.2";
      =     L 0.1;
      A     L 0.1;
      AN    "LOCK_DOORS_RELAY";
      S     "LOCK_DOORS_RELAY";
      =     "M1008.1";
      A     L 0.1;
      AN    "M1008.1";
      A     "LOCK_DOORS_RELAY";
      R     "LOCK_DOORS_RELAY";
      A     L 0.0;
      A     "LOCK_DOORS_RELAY";
      A(;
      O     "E2.1";
      O;
      AN    "E2.1";
      A     "Clock 0.5 S";
      );
      =     "Lamp_Door_Locked";
NETWORK
TITLE = Simodrive Reset realy
      AN    "Bypass";
      =     "SIMODRIVE_RESET";
NETWORK
TITLE = Table locker cylinder up
      A(;
      O     "M32.5";
      O     "M53.0";
      );
      AN    "FWD_TABLE_ROTATION";
      AN    "REVERSE_TABLE_ROTATION";
      =     "Table locker cylinder up";
NETWORK
TITLE = Table locker cylinder down
      A(;
      O     "M32.4";
      O     "M42.1";
      O     "M53.1";
      );
      AN    "FWD_TABLE_ROTATION";
      AN    "REVERSE_TABLE_ROTATION";
      =     "TABLE_LCKER_DWN";
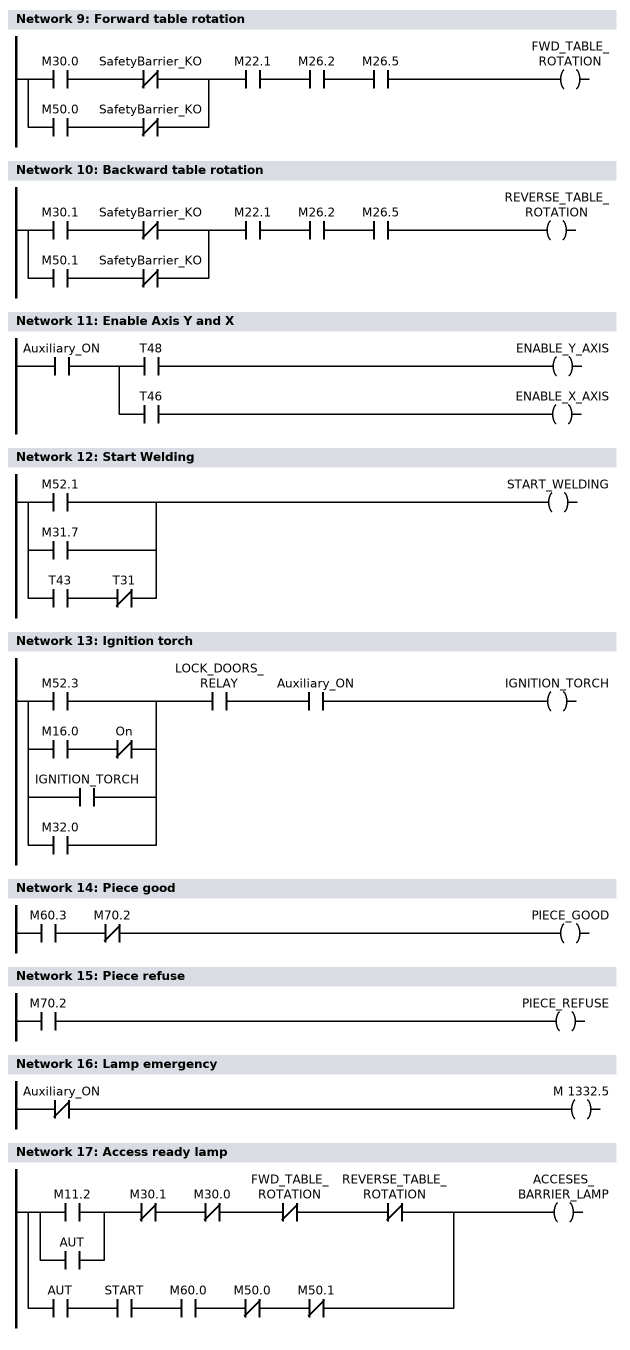
NETWORK
TITLE = Forward table rotation
      A(;
      A     "M30.0";
      AN    "SafetyBarrier_KO";
      O;
      A     "M50.0";
      AN    "SafetyBarrier_KO";
      );
      A     "M22.1";
      A     "M26.2";
      A     "M26.5";
      =     "FWD_TABLE_ROTATION";
NETWORK
TITLE = Backward table rotation
      A(;
      A     "M30.1";
      AN    "SafetyBarrier_KO";
      O;
      A     "M50.1";
      AN    "SafetyBarrier_KO";
      );
      A     "M22.1";
      A     "M26.2";
      A     "M26.5";
      =     "REVERSE_TABLE_ROTATION";
NETWORK
TITLE = Enable Axis Y and X
      A     "Auxiliary_ON";
      =     L 0.0;
      A     L 0.0;
      A     "T48";
      =     "ENABLE_Y_AXIS";
      A     L 0.0;
      A     "T46";
      =     "ENABLE_X_AXIS";
NETWORK
TITLE = Start Welding
      O     "M52.1";
      O     "M31.7";
      O;
      A     "T43";
      AN    "T31";
      =     "START_WELDING";
NETWORK
TITLE = Ignition torch
      A(;
      O     "M52.3";
      O;
      A     "M16.0";
      AN    "On";
      O     "IGNITION_TORCH";
      O     "M32.0";
      );
      A     "LOCK_DOORS_RELAY";
      A     "Auxiliary_ON";
      =     "IGNITION_TORCH";
NETWORK
TITLE = Piece good
      A     "M60.3";
      AN    "M70.2";
      =     "PIECE_GOOD";
NETWORK
TITLE = Piece refuse
      A     "M70.2";
      =     "PIECE_REFUSE";
NETWORK
TITLE = Lamp emergency
      AN    "Auxiliary_ON";
      =     M 1332.5;
NETWORK
TITLE = Access ready lamp
      A(;
      O     "M11.2";
      O     "AUT";
      );
      AN    "M30.1";
      AN    "M30.0";
      AN    "FWD_TABLE_ROTATION";
      AN    "REVERSE_TABLE_ROTATION";
      O;
      A     "AUT";
      A     "START";
      A     "M60.0";
      AN    "M50.0";
      AN    "M50.1";
      =     "ACCESES_BARRIER_LAMP";
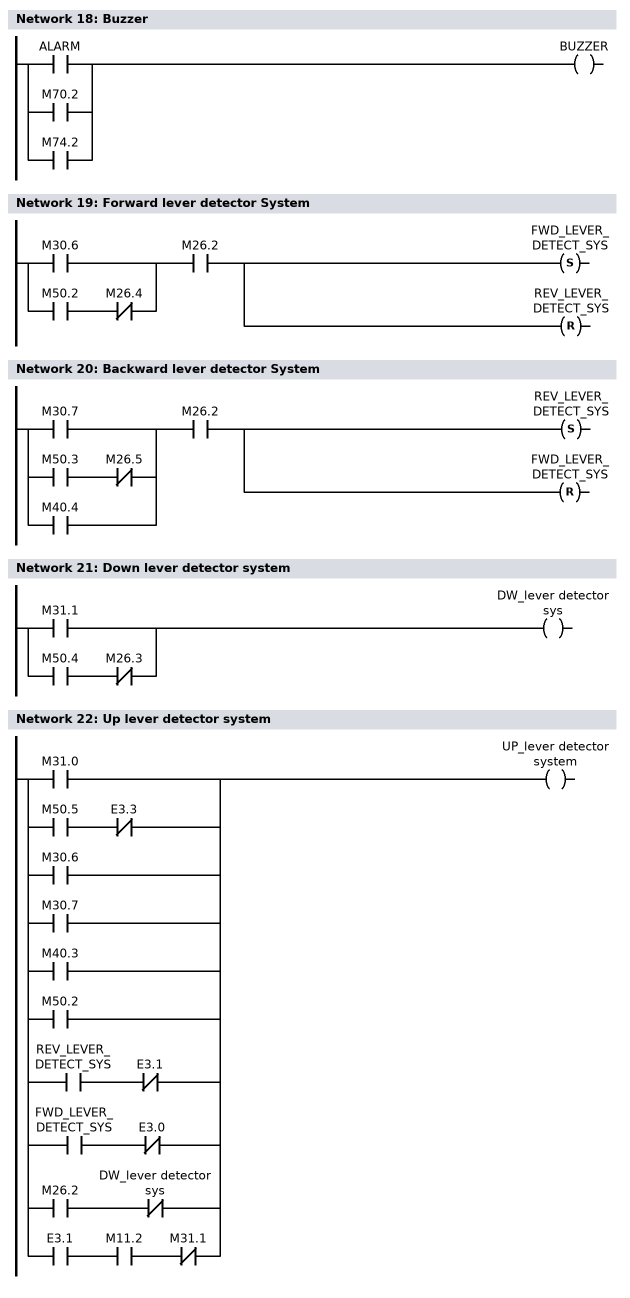
NETWORK
TITLE = Buzzer
//"Off"
      O     "ALARM";
      O     "M70.2";
      O     "M74.2";
      =     "BUZZER";
NETWORK
TITLE = Forward lever detector System
      A(;
      O     "M30.6";
      O;
      A     "M50.2";
      AN    "M26.4";
      );
      A     "M26.2";
      S     "FWD_LEVER_DETECT_SYS";
      R     "REV_LEVER_DETECT_SYS";
NETWORK
TITLE = Backward lever detector System
      A(;
      O     "M30.7";
      O;
      A     "M50.3";
      AN    "M26.5";
      O     "M40.4";
      );
      A     "M26.2";
      S     "REV_LEVER_DETECT_SYS";
      R     "FWD_LEVER_DETECT_SYS";
NETWORK
TITLE = Down lever detector system
      O     "M31.1";
      O;
      A     "M50.4";
      AN    "M26.3";
      =     "DW_lever detector sys";
NETWORK
TITLE = Up lever detector system
      O     "M31.0";
      O;
      A     "M50.5";
      AN    "E3.3";
      O     "M30.6";
      O     "M30.7";
      O     "M40.3";
      O     "M50.2";
      O;
      A     "REV_LEVER_DETECT_SYS";
      AN    "E3.1";
      O;
      A     "FWD_LEVER_DETECT_SYS";
      AN    "E3.0";
      O;
      A     "M26.2";
      AN    "DW_lever detector sys";
      O;
      A     "E3.1";
      A     "M11.2";
      AN    "M31.1";
      =     "UP_lever detector system";
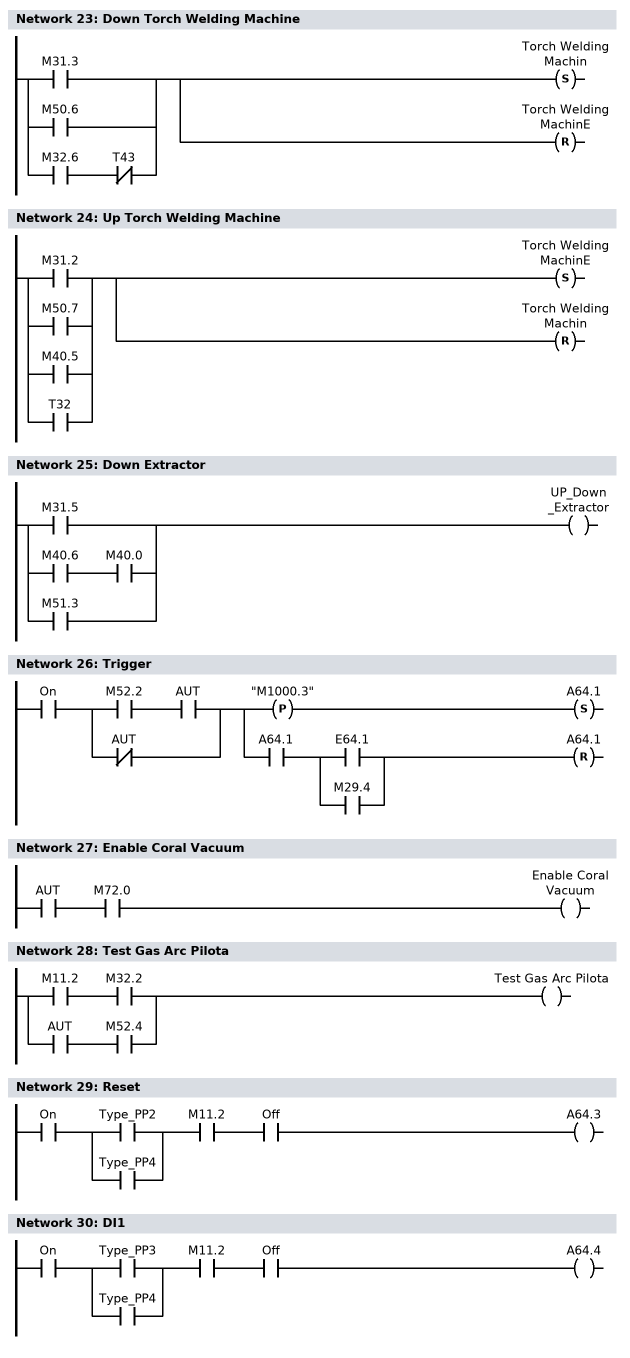
NETWORK
TITLE = Down Torch Welding Machine
      O     "M31.3";
      O     "M50.6";
      O;
      A     "M32.6";
      AN    "T43";
      S     "Torch Welding Machin";
      R     "Torch Welding MachinE";
NETWORK
TITLE = Up Torch Welding Machine
      O     "M31.2";
      O     "M50.7";
      O     "M40.5";
      O     "T32";
      S     "Torch Welding MachinE";
      R     "Torch Welding Machin";
NETWORK
TITLE = Down Extractor
      O     "M31.5";
      O;
      A     "M40.6";
      A     "M40.0";
      O     "M51.3";
      =     "UP_Down _Extractor";
NETWORK
TITLE = Trigger
      A     "On";
      A(;
      A     "M52.2";
      A     "AUT";
      ON    "AUT";
      );
      =     L 0.0;
      A     L 0.0;
      FP    "M1000.3";
      S     "A64.1";
      A     L 0.0;
      A     "A64.1";
      A(;
      O     "E64.1";
      O     "M29.4";
      );
      R     "A64.1";
NETWORK
TITLE = Enable Coral Vacuum
      A     "AUT";
      A     "M72.0";
      =     "Enable Coral Vacuum";
NETWORK
TITLE = Test Gas Arc Pilota
//Test Arco Gas
      A     "M11.2";
      A     "M32.2";
      O;
      A     "AUT";
      A     "M52.4";
      =     "Test Gas Arc Pilota";
NETWORK
TITLE = Reset
//bit DI0 Select Scene TeleCam
      A     "On";
      A(;
      O     "Type_PP2";
      O     "Type_PP4";
      );
      A     "M11.2";
      A     "Off";
      =     "A64.3";
NETWORK
TITLE = DI1
//bit DI1 Select Scene TeleCam
      A     "On";
      A(;
      O     "Type_PP3";
      O     "Type_PP4";
      );
      A     "M11.2";
      A     "Off";
      =     "A64.4";
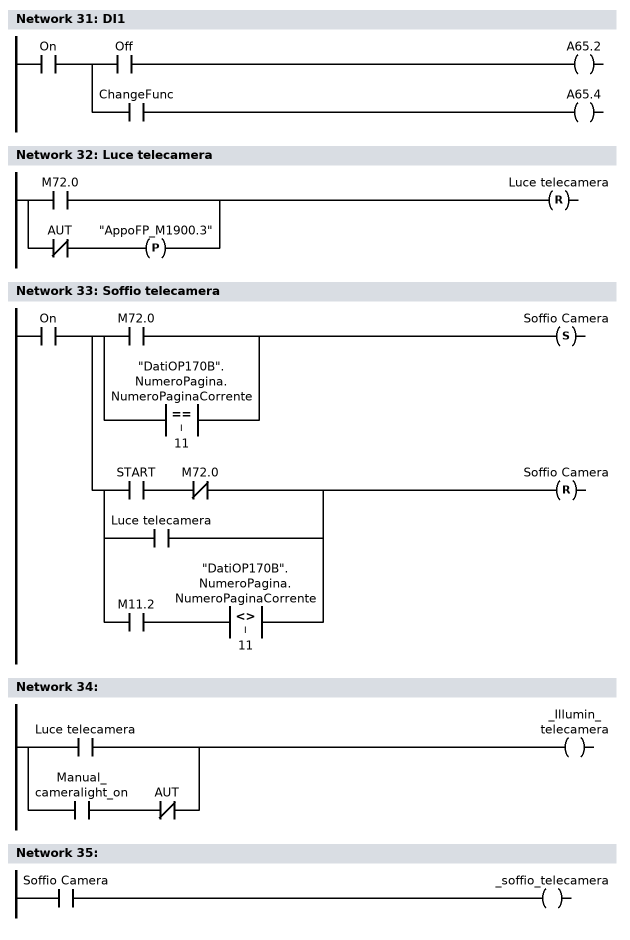
NETWORK
TITLE = DI1
//Select Scene Cam
      A     "On";
      =     L 0.0;
      A     L 0.0;
      A     "Off";
      =     "A65.2";
      A     L 0.0;
      A     "ChangeFunc";
      =     "A65.4";
NETWORK
TITLE = Luce telecamera
      O     "M72.0";
      O(;
      AN    "AUT";
      FP    "AppoFP_M1900.3";
      );
      R     "Luce telecamera";
NETWORK
TITLE = Soffio telecamera
      A     "On";
      =     L 0.0;
      A     L 0.0;
      A(;
      O     "M72.0";
      O(;
      L     "DatiOP170B".NumeroPagina.NumeroPaginaCorrente;
      L     11;
      ==I;
      );
      );
      S     "Soffio Camera";
      A     L 0.0;
      A(;
      A     "START";
      AN    "M72.0";
      O     "Luce telecamera";
      O;
      A     "M11.2";
      A(;
      L     "DatiOP170B".NumeroPagina.NumeroPaginaCorrente;
      L     11;
      <>I;
      );
      );
      R     "Soffio Camera";
NETWORK
TITLE =
      O     "Luce telecamera";
      O;
      A     "Manual_cameralight_on";
      AN    "AUT";
      =     "_Illumin_telecamera";
NETWORK
TITLE =
      A     "Soffio Camera";
      =     "_soffio_telecamera";
END_FUNCTION

FUNCTION "FC19 - REPOSITIONING" : VOID	// FC 19
TITLE = Repositioning management
VERSION : 0.1
BEGIN
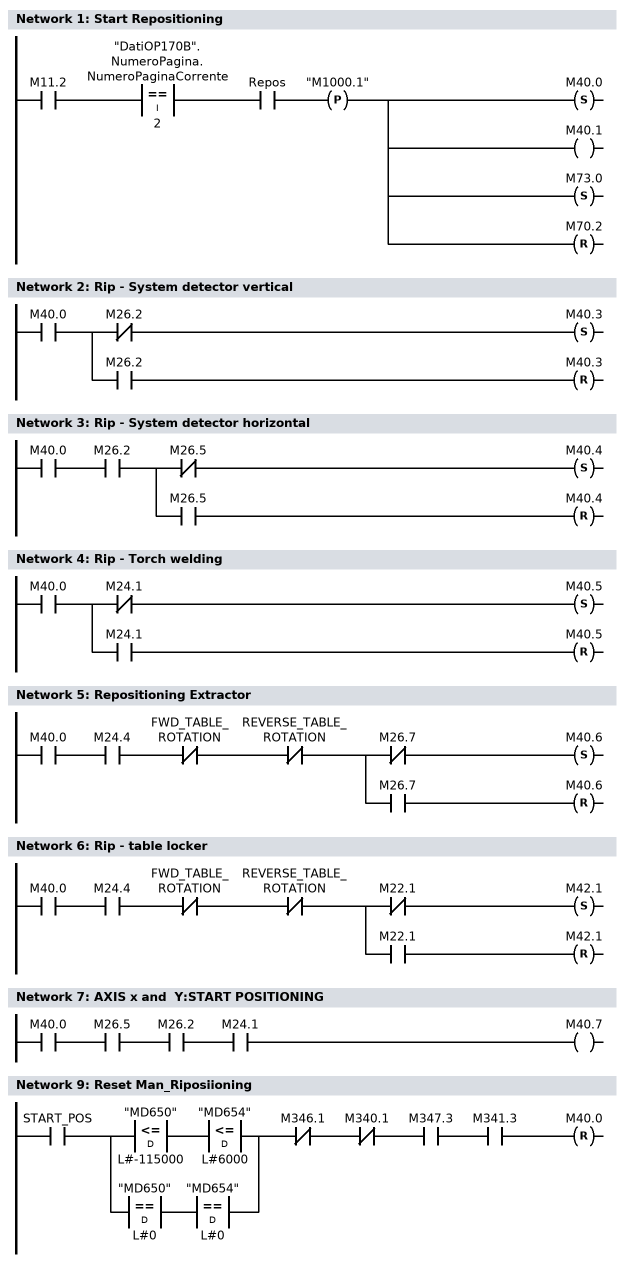
NETWORK
TITLE = Start Repositioning
      A     "M11.2";
      A(;
      L     "DatiOP170B".NumeroPagina.NumeroPaginaCorrente;
      L     2;
      ==I;
      );
      A     "Repos";
      FP    "M1000.1";
      S     "M40.0";
      =     "M40.1";
      S     "M73.0";
      R     "M70.2";
NETWORK
TITLE = Rip - System detector vertical
//ripositioning Table
      A     "M40.0";
      =     L 0.0;
      A     L 0.0;
      AN    "M26.2";
      S     "M40.3";
      A     L 0.0;
      A     "M26.2";
      R     "M40.3";
NETWORK
TITLE = Rip - System detector horizontal
//ripositioning Table
      A     "M40.0";
      A     "M26.2";
      =     L 0.0;
      A     L 0.0;
      AN    "M26.5";
      S     "M40.4";
      A     L 0.0;
      A     "M26.5";
      R     "M40.4";
NETWORK
TITLE = Rip - Torch welding
//ripositioning Table
      A     "M40.0";
      =     L 0.0;
      A     L 0.0;
      AN    "M24.1";
      S     "M40.5";
      A     L 0.0;
      A     "M24.1";
      R     "M40.5";
NETWORK
TITLE = Repositioning Extractor
      A     "M40.0";
      A     "M24.4";
      AN    "FWD_TABLE_ROTATION";
      AN    "REVERSE_TABLE_ROTATION";
      =     L 0.0;
      A     L 0.0;
      AN    "M26.7";
      S     "M40.6";
      A     L 0.0;
      A     "M26.7";
      R     "M40.6";
NETWORK
TITLE = Rip - table locker
      A     "M40.0";
      A     "M24.4";
      AN    "FWD_TABLE_ROTATION";
      AN    "REVERSE_TABLE_ROTATION";
      =     L 0.0;
      A     L 0.0;
      AN    "M22.1";
      S     "M42.1";
      A     L 0.0;
      A     "M22.1";
      R     "M42.1";
NETWORK
TITLE = AXIS x and  Y:START POSITIONING
      A     "M40.0";
      A     "M26.5";
      A     "M26.2";
      A     "M24.1";
      =     "M40.7";
NETWORK
TITLE = Reset Man_Riposiioning
//      U     "START_POS"
//      U(    
//      U(    
//      L     "MD650"
//      L     L#-115000
//      <=D   
//      )     
//      U(    
//      L     "MD654"
//      L     L#6000
//      <=D   
//      )     
//      O     
//      U(    
//      L     "MD650"
//      L     L#0
//      ==I   
//      )     
//      U(    
//      L     "MD654"
//      L     L#0
//      ==I   
//      )     
//      )     
//      UN    "M346.1"
//      UN    "M340.1"
//      U     "M347.3"
//      U     "M341.3"
//      R     "M40.0"
NETWORK
TITLE = Reset Man_Riposiioning
      A     "START_POS";
      A(;
      A(;
      L     "MD650";
      L     L#-115000;
      <=D;
      );
      A(;
      L     "MD654";
      L     L#6000;
      <=D;
      );
      O;
      A(;
      L     "MD650";
      L     L#0;
      ==D;
      );
      A(;
      L     "MD654";
      L     L#0;
      ==D;
      );
      );
      AN    "M346.1";
      AN    "M340.1";
      A     "M347.3";
      A     "M341.3";
      R     "M40.0";
NETWORK
TITLE =
END_FUNCTION

FUNCTION "FC50 - TEACH-IN" : VOID	// FC 50
TITLE = TEACH_IN
VERSION : 0.1
BEGIN
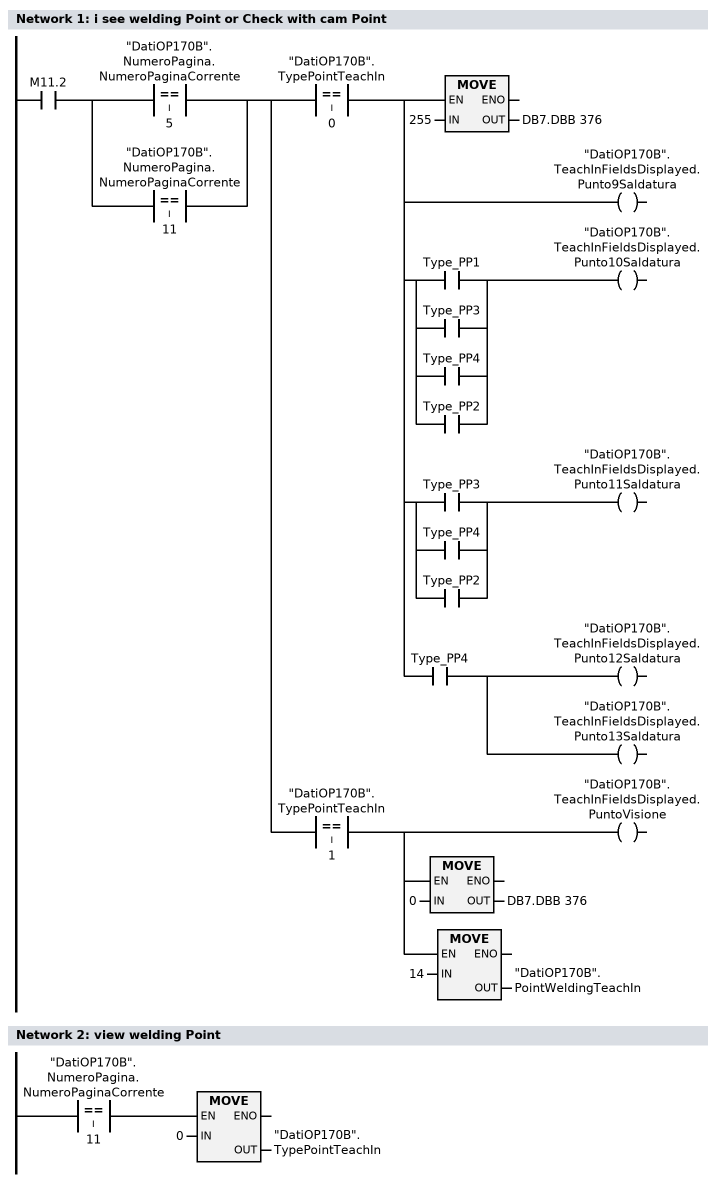
NETWORK
TITLE = i see welding Point or Check with cam Point
      A     "M11.2";
      A(;
      O(;
      L     "DatiOP170B".NumeroPagina.NumeroPaginaCorrente;
      L     5;
      ==I;
      );
      O(;
      L     "DatiOP170B".NumeroPagina.NumeroPaginaCorrente;
      L     11;
      ==I;
      );
      );
      =     L 0.0;
      A     L 0.0;
      A(;
      L     "DatiOP170B".TypePointTeachIn;
      L     0;
      ==I;
      );
      =     L 0.1;
      A     L 0.1;
      JNB   _001;
      L     255;
      T     DB7.DBB 376;
_001: NOP   0;
      A     L 0.1;
      BLD   102;
      =     "DatiOP170B".TeachInFieldsDisplayed.Punto9Saldatura;
      A     L 0.1;
      A(;
      O     "Type_PP1";
      O     "Type_PP3";
      O     "Type_PP4";
      O     "Type_PP2";
      );
      =     "DatiOP170B".TeachInFieldsDisplayed.Punto10Saldatura;
      A     L 0.1;
      A(;
      O     "Type_PP3";
      O     "Type_PP4";
      O     "Type_PP2";
      );
      =     "DatiOP170B".TeachInFieldsDisplayed.Punto11Saldatura;
      A     L 0.1;
      A     "Type_PP4";
      =     "DatiOP170B".TeachInFieldsDisplayed.Punto12Saldatura;
      =     "DatiOP170B".TeachInFieldsDisplayed.Punto13Saldatura;
      A     L 0.0;
      A(;
      L     "DatiOP170B".TypePointTeachIn;
      L     1;
      ==I;
      );
      =     L 0.1;
      A     L 0.1;
      BLD   102;
      =     "DatiOP170B".TeachInFieldsDisplayed.PuntoVisione;
      A     L 0.1;
      JNB   _002;
      L     0;
      T     DB7.DBB 376;
_002: NOP   0;
      A     L 0.1;
      JNB   _003;
      L     14;
      T     "DatiOP170B".PointWeldingTeachIn;
_003: NOP   0;
NETWORK
TITLE = view welding Point
      A(;
      L     "DatiOP170B".NumeroPagina.NumeroPaginaCorrente;
      L     11;
      ==I;
      );
      JNB   _004;
      L     0;
      T     "DatiOP170B".TypePointTeachIn;
_004: NOP   0;
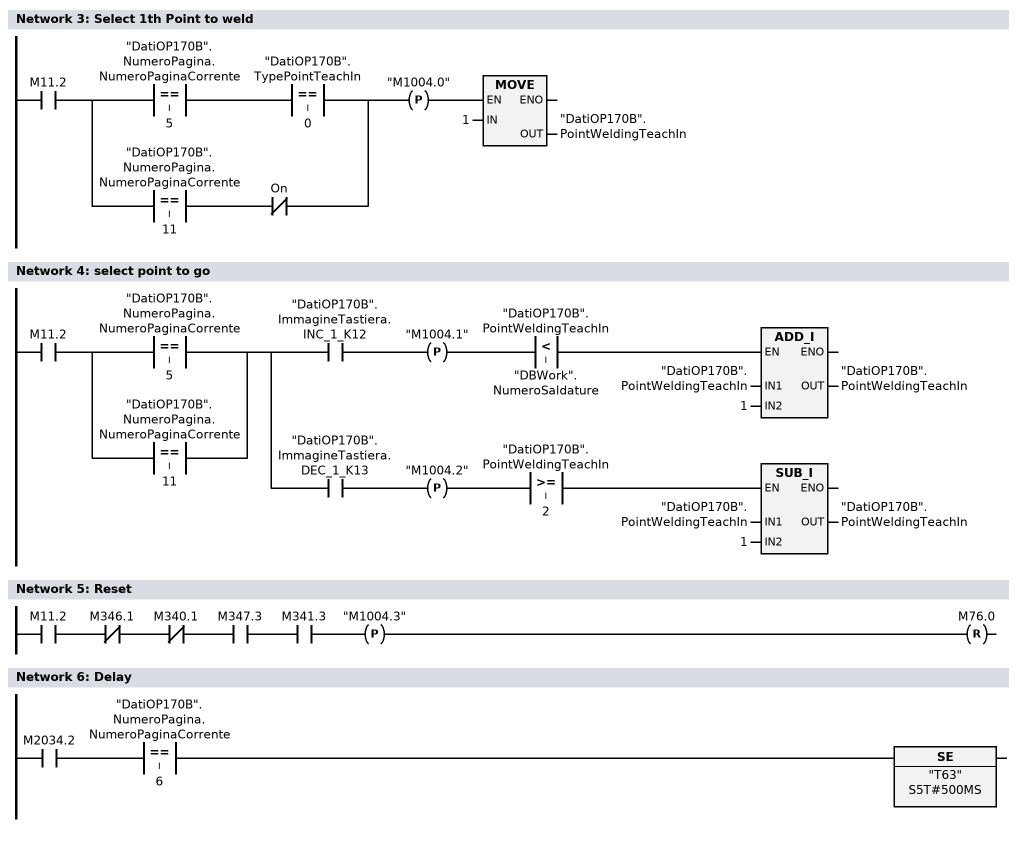
NETWORK
TITLE = Select 1th Point to weld
      A     "M11.2";
      A(;
      A(;
      L     "DatiOP170B".NumeroPagina.NumeroPaginaCorrente;
      L     5;
      ==I;
      );
      A(;
      L     "DatiOP170B".TypePointTeachIn;
      L     0;
      ==I;
      );
      O;
      A(;
      L     "DatiOP170B".NumeroPagina.NumeroPaginaCorrente;
      L     11;
      ==I;
      );
      AN    "On";
      );
      FP    "M1004.0";
      JNB   _005;
      L     1;
      T     "DatiOP170B".PointWeldingTeachIn;
_005: NOP   0;
NETWORK
TITLE = select point to go
      A     "M11.2";
      A(;
      O(;
      L     "DatiOP170B".NumeroPagina.NumeroPaginaCorrente;
      L     5;
      ==I;
      );
      O(;
      L     "DatiOP170B".NumeroPagina.NumeroPaginaCorrente;
      L     11;
      ==I;
      );
      );
      =     L 0.0;
      A     L 0.0;
      A     "DatiOP170B".ImmagineTastiera.INC_1_K12;
      FP    "M1004.1";
      A(;
      L     "DatiOP170B".PointWeldingTeachIn;
      L     "DBWork".NumeroSaldature;
      <I;
      );
      JNB   _006;
      L     "DatiOP170B".PointWeldingTeachIn;
      L     1;
      +I;
      T     "DatiOP170B".PointWeldingTeachIn;
_006: NOP   0;
      A     L 0.0;
      A     "DatiOP170B".ImmagineTastiera.DEC_1_K13;
      FP    "M1004.2";
      A(;
      L     "DatiOP170B".PointWeldingTeachIn;
      L     2;
      >=I;
      );
      JNB   _007;
      L     "DatiOP170B".PointWeldingTeachIn;
      L     1;
      -I;
      T     "DatiOP170B".PointWeldingTeachIn;
_007: NOP   0;
NETWORK
TITLE = Reset
      A     "M11.2";
      AN    "M346.1";
      AN    "M340.1";
      A     "M347.3";
      A     "M341.3";
      FP    "M1004.3";
      R     "M76.0";
NETWORK
TITLE = Delay
      A     "M2034.2";
      A(;
      L     "DatiOP170B".NumeroPagina.NumeroPaginaCorrente;
      L     6;
      ==I;
      );
      L     S5T#500MS;
      SE    "T63";
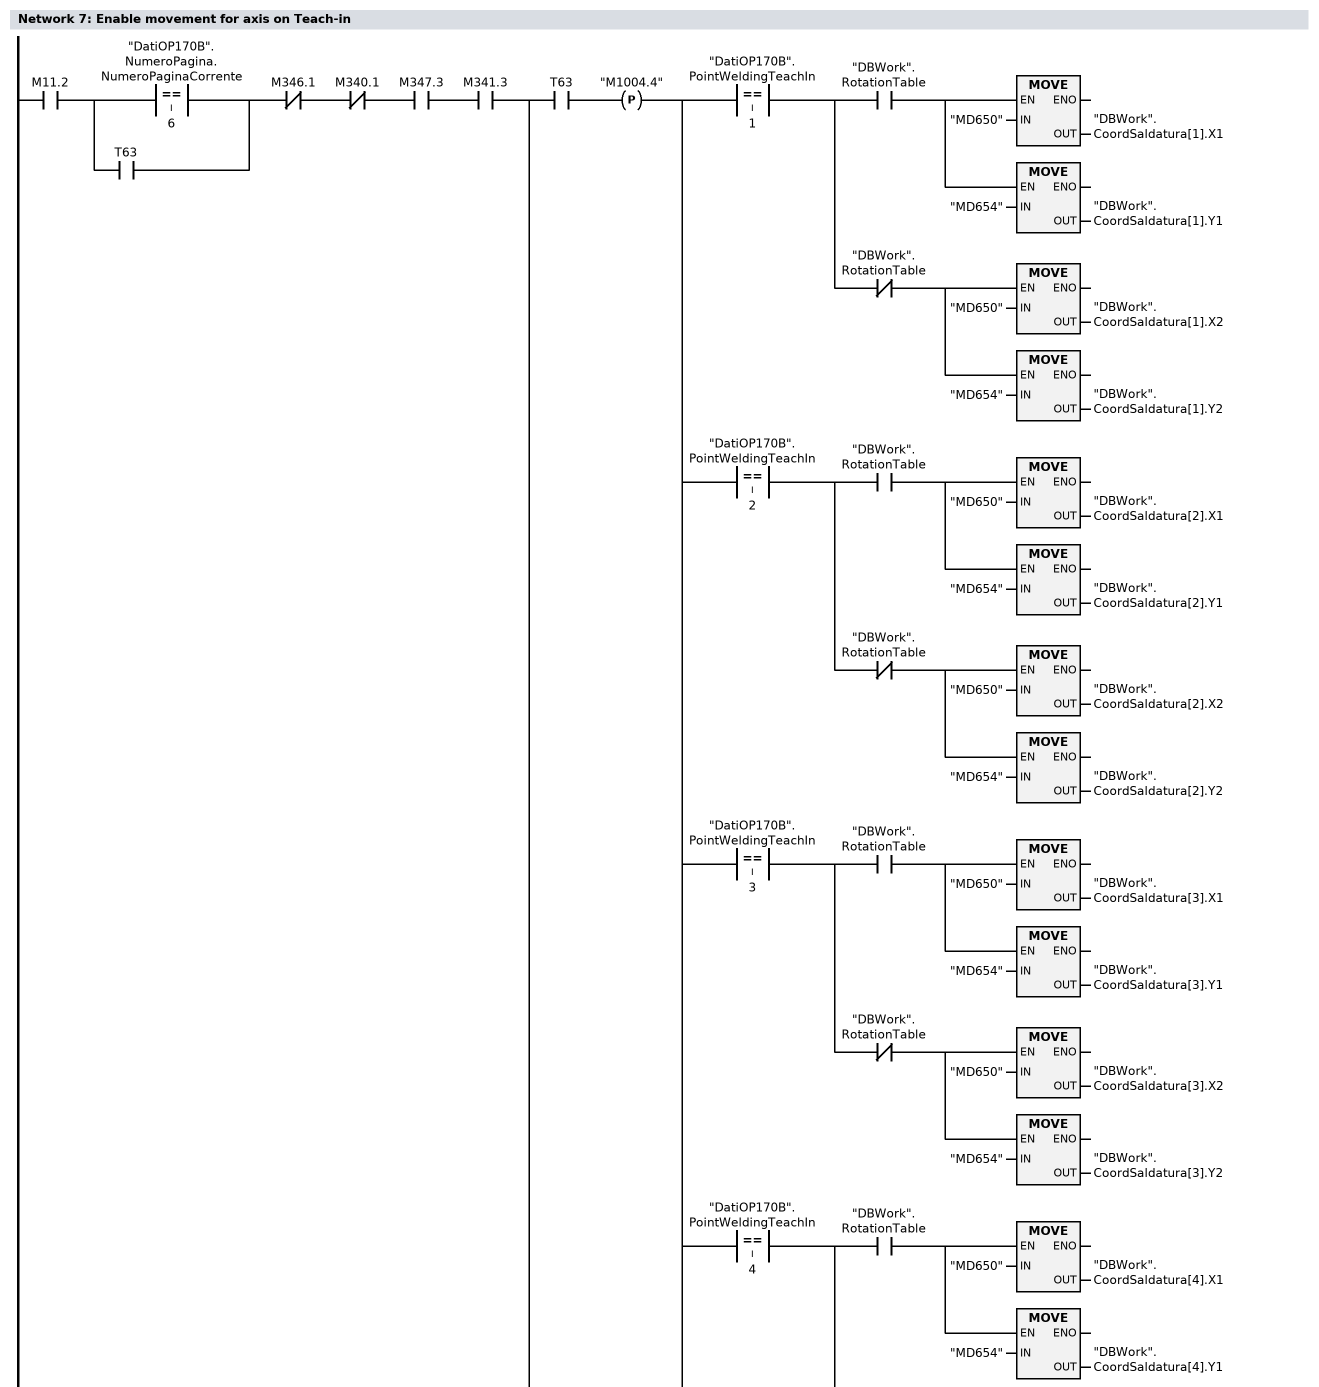
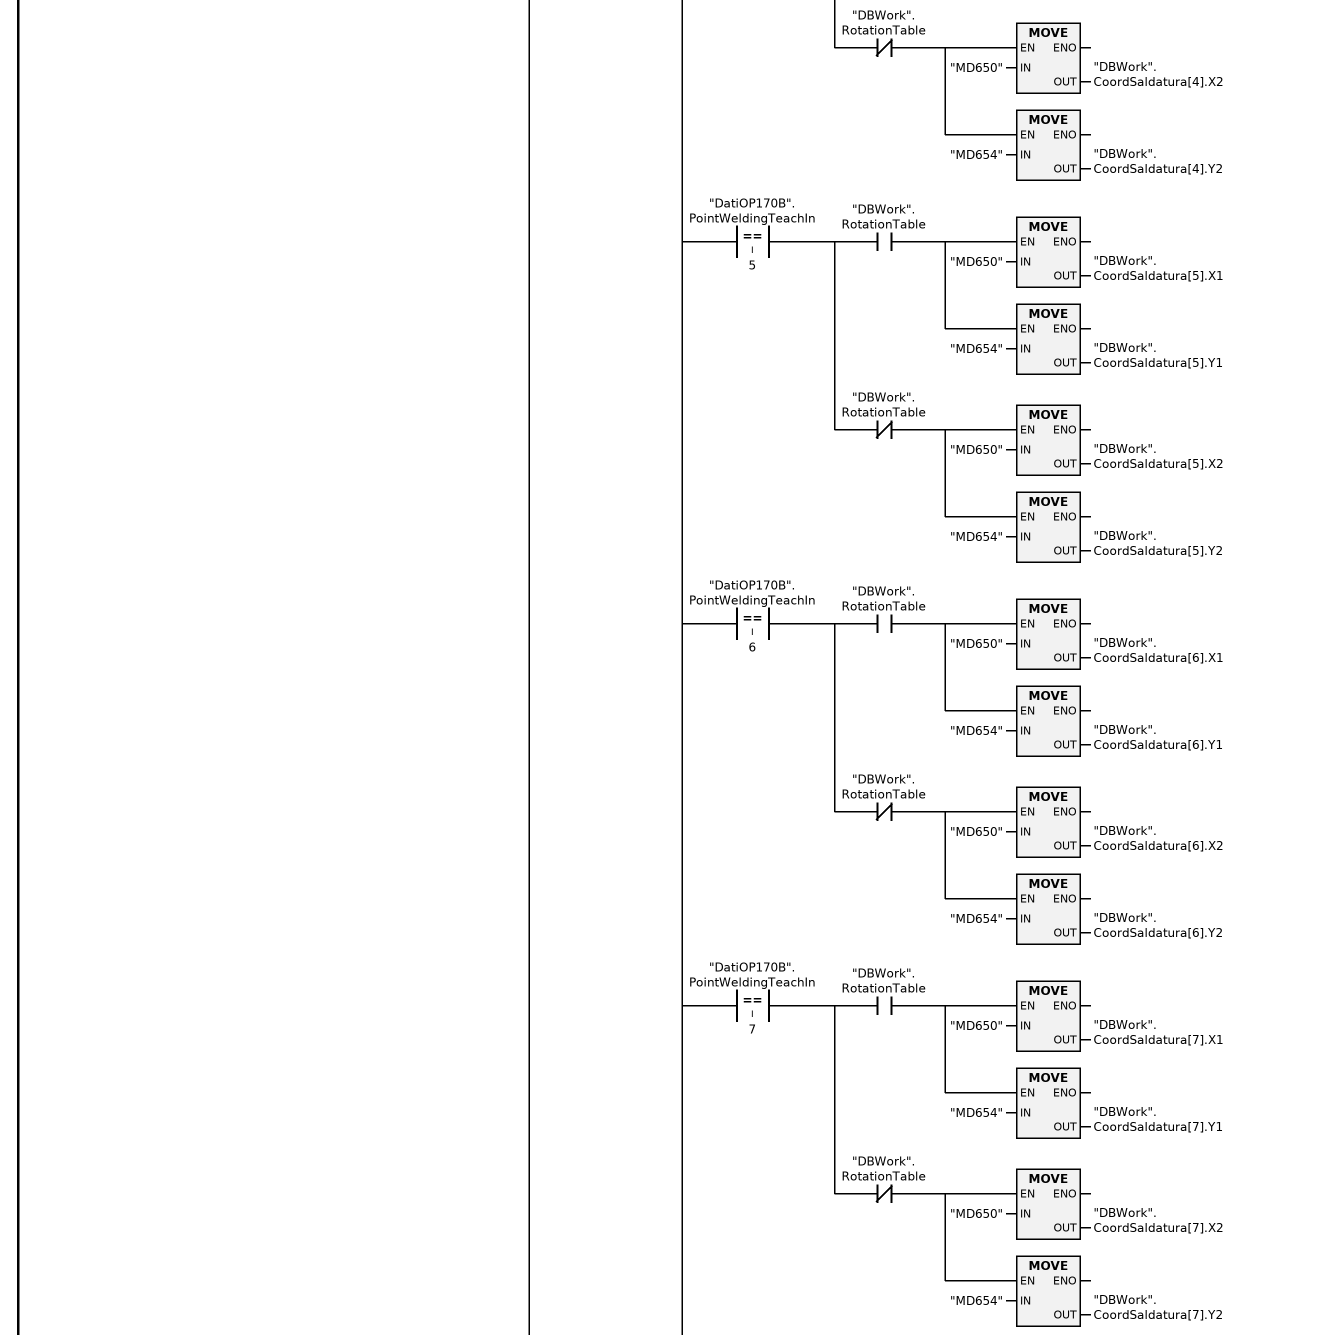
